LIN {X 0,Y 518.293,Z 267.839,A -85,B 0,C 180,E1 -4920.11,E2 -4920.11} C_VEL
LIN {X 0,Y 518.366,Z 255.687,A -85,B 0,C 180,E1 -4920.557,E2 -4920.557} C_VEL
LIN {X 0,Y 516.298,Z 245.529,A -85,B 0,C 180,E1 -4920.881,E2 -4920.881} C_VEL
LIN {X 0,Y 516.387,Z 241.725,A -85,B 0,C 180,E1 -4924.182,E2 -4924.182} C_VEL
LIN {X 0,Y 516.405,Z 238.771,A -85,B 0,C 180,E1 -4926.755,E2 -4926.755} C_VEL
LIN {X 0,Y 516.418,Z 234.973,A -85,B 0,C 180,E1 -4930.11,E2 -4930.11} C_VEL
LIN {X 0,Y 516.464,Z 232.179,A -85,B 0,C 180,E1 -4932.581,E2 -4932.581} C_VEL
LIN {X 0,Y 516.496,Z 228.529,A -85,B 0,C 180,E1 -4935.823,E2 -4935.823} C_VEL
LIN {X 0,Y 516.609,Z 224.947,A -85,B 0,C 180,E1 -4939.021,E2 -4939.021} C_VEL
LIN {X 0,Y 516.557,Z 224.144,A -85,B 0,C 180,E1 -4939.813,E2 -4939.813} C_VEL
LIN {X 0,Y 516.894,Z 224.101,A -85,B 0,C 180,E1 -4942.186,E2 -4942.186} C_VEL
LIN {X 0,Y 517.03,Z 224.083,A -85,B 0,C 180,E1 -4944.54,E2 -4944.54} C_VEL
LIN {X 0,Y 517.069,Z 224.078,A -85,B 0,C 180,E1 -4947.664,E2 -4947.664} C_VEL
LIN {X 0,Y 517.082,Z 224.079,A -85,B 0,C 180,E1 -4950.779,E2 -4950.779} C_VEL
LIN {X 0,Y 517.001,Z 224.089,A -85,B 0,C 180,E1 -4953.117,E2 -4953.117} C_VEL
LIN {X 0,Y 516.996,Z 224.086,A -85,B 0,C 180,E1 -4956.244,E2 -4956.244} C_VEL
LIN {X 0,Y 516.943,Z 224.094,A -85,B 0,C 180,E1 -4959.39,E2 -4959.39} C_VEL
LIN {X 0,Y 516.967,Z 224.089,A -85,B 0,C 180,E1 -4961.825,E2 -4961.825} C_VEL
LIN {X 0,Y 516.928,Z 224.097,A -85,B 0,C 180,E1 -4965.147,E2 -4965.147} C_VEL
LIN {X 0,Y 516.912,Z 224.097,A -85,B 0,C 180,E1 -4968.223,E2 -4968.223} C_VEL
LIN {X 0,Y 516.902,Z 224.1,A -85,B 0,C 180,E1 -4970.702,E2 -4970.702} C_VEL
LIN {X 0,Y 516.881,Z 224.104,A -85,B 0,C 180,E1 -4973.223,E2 -4973.223} C_VEL
LIN {X 0,Y 516.932,Z 224.095,A -85,B 0,C 180,E1 -4976.198,E2 -4976.198} C_VEL
LIN {X 0,Y 516.909,Z 224.099,A -85,B 0,C 180,E1 -4979.306,E2 -4979.306} C_VEL
LIN {X 0,Y 516.889,Z 224.101,A -85,B 0,C 180,E1 -4982.546,E2 -4982.546} C_VEL
LIN {X 0,Y 516.871,Z 224.103,A -85,B 0,C 180,E1 -4985.334,E2 -4985.334} C_VEL
LIN {X 0,Y 516.871,Z 224.103,A -85,B 0,C 180,E1 -4987.945,E2 -4987.945} C_VEL
LIN {X 0,Y 516.898,Z 224.1,A -85,B 0,C 180,E1 -4990.741,E2 -4990.741} C_VEL
LIN {X 0,Y 516.873,Z 224.103,A -85,B 0,C 180,E1 -4993.904,E2 -4993.904} C_VEL
LIN {X 0,Y 516.873,Z 224.104,A -85,B 0,C 180,E1 -4996.108,E2 -4996.108} C_VEL
LIN {X 0,Y 516.896,Z 224.101,A -85,B 0,C 180,E1 -4999.262,E2 -4999.262} C_VEL
LIN {X 0,Y 516.875,Z 224.104,A -85,B 0,C 180,E1 -5002.058,E2 -5002.058} C_VEL
LIN {X 0,Y 516.888,Z 224.101,A -85,B 0,C 180,E1 -5005.178,E2 -5005.178} C_VEL
LIN {X 0,Y 516.878,Z 224.104,A -85,B 0,C 180,E1 -5007.977,E2 -5007.977} C_VEL
LIN {X 0,Y 516.932,Z 224.095,A -85,B 0,C 180,E1 -5010.698,E2 -5010.698} C_VEL
LIN {X 0,Y 516.939,Z 224.096,A -85,B 0,C 180,E1 -5013.805,E2 -5013.805} C_VEL
LIN {X 0,Y 516.869,Z 224.102,A -85,B 0,C 180,E1 -5016.778,E2 -5016.778} C_VEL
LIN {X 0,Y 516.937,Z 224.096,A -85,B 0,C 180,E1 -5019.733,E2 -5019.733} C_VEL
LIN {X 0,Y 516.93,Z 224.095,A -85,B 0,C 180,E1 -5022.598,E2 -5022.598} C_VEL
LIN {X 0,Y 516.941,Z 224.093,A -85,B 0,C 180,E1 -5025.032,E2 -5025.032} C_VEL
LIN {X 0,Y 516.966,Z 224.092,A -85,B 0,C 180,E1 -5028.235,E2 -5028.235} C_VEL
LIN {X 0,Y 516.955,Z 224.092,A -85,B 0,C 180,E1 -5031.401,E2 -5031.401} C_VEL
LIN {X 0,Y 517.011,Z 224.086,A -85,B 0,C 180,E1 -5033.758,E2 -5033.758} C_VEL
LIN {X 0,Y 517.082,Z 224.079,A -85,B 0,C 180,E1 -5037.664,E2 -5037.664} C_VEL
LIN {X 0,Y 517.094,Z 224.074,A -85,B 0,C 180,E1 -5040.78,E2 -5040.78} C_VEL
LIN {X 0,Y 517.013,Z 224.084,A -85,B 0,C 180,E1 -5043.118,E2 -5043.118} C_VEL
LIN {X 0,Y 516.992,Z 224.087,A -85,B 0,C 180,E1 -5046.245,E2 -5046.245} C_VEL
LIN {X 0,Y 516.945,Z 224.095,A -85,B 0,C 180,E1 -5049.391,E2 -5049.391} C_VEL
LIN {X 0,Y 516.956,Z 224.094,A -85,B 0,C 180,E1 -5051.808,E2 -5051.808} C_VEL
LIN {X 0,Y 516.95,Z 224.093,A -85,B 0,C 180,E1 -5055.147,E2 -5055.147} C_VEL
LIN {X 0,Y 516.93,Z 224.094,A -85,B 0,C 180,E1 -5058.223,E2 -5058.223} C_VEL
LIN {X 0,Y 516.918,Z 224.097,A -85,B 0,C 180,E1 -5060.702,E2 -5060.702} C_VEL
LIN {X 0,Y 516.891,Z 224.1,A -85,B 0,C 180,E1 -5064.074,E2 -5064.074} C_VEL
LIN {X 0,Y 516.915,Z 224.097,A -85,B 0,C 180,E1 -5066.659,E2 -5066.659} C_VEL
LIN {X 0,Y 516.915,Z 224.098,A -85,B 0,C 180,E1 -5069.524,E2 -5069.524} C_VEL
LIN {X 0,Y 516.9,Z 224.099,A -85,B 0,C 180,E1 -5072.544,E2 -5072.544} C_VEL
LIN {X 0,Y 516.872,Z 224.103,A -85,B 0,C 180,E1 -5075.33,E2 -5075.33} C_VEL
LIN {X 0,Y 516.886,Z 224.102,A -85,B 0,C 180,E1 -5077.943,E2 -5077.943} C_VEL
LIN {X 0,Y 516.889,Z 224.102,A -85,B 0,C 180,E1 -5080.742,E2 -5080.742} C_VEL
LIN {X 0,Y 516.888,Z 224.101,A -85,B 0,C 180,E1 -5082.832,E2 -5082.832} C_VEL
LIN {X 0,Y 516.901,Z 224.098,A -85,B 0,C 180,E1 -5085.007,E2 -5085.007} C_VEL
LIN {X 0,Y 516.919,Z 224.097,A -85,B 0,C 180,E1 -5088.399,E2 -5088.399} C_VEL
LIN {X 0,Y 516.919,Z 224.183,A -85,B 0,C 180,E1 -5091.168,E2 -5091.168} C_VEL
LIN {X 0,Y 518.071,Z 230.899,A -85,B 0,C 180,E1 -5093.835,E2 -5093.835} C_VEL
LIN {X 0,Y 518.092,Z 236.578,A -85,B 0,C 180,E1 -5095.841,E2 -5095.841} C_VEL
LIN {X 0,Y 517.808,Z 245.682,A -85,B 0,C 180,E1 -5098.952,E2 -5098.952} C_VEL
LIN {X 0,Y 517.592,Z 254.692,A -85,B 0,C 180,E1 -5101.957,E2 -5101.957} C_VEL
LIN {X 0,Y 517.295,Z 264.28,A -85,B 0,C 180,E1 -5105.091,E2 -5105.091} C_VEL
LIN {X 0,Y 517.075,Z 273.548,A -85,B 0,C 180,E1 -5108.051,E2 -5108.051} C_VEL
LIN {X 0,Y 516.883,Z 282.815,A -85,B 0,C 180,E1 -5110.954,E2 -5110.954} C_VEL
LIN {X 0,Y 516.697,Z 292.082,A -85,B 0,C 180,E1 -5113.809,E2 -5113.809} C_VEL
LIN {X 0,Y 516.588,Z 299.708,A -85,B 0,C 180,E1 -5116.095,E2 -5116.095} C_VEL
LIN {X 0,Y 518.517,Z 312.169,A -85,B 0,C 180,E1 -5116.428,E2 -5116.428} C_VEL
LIN {X 0,Y 518.247,Z 324.975,A -85,B 0,C 180,E1 -5116.87,E2 -5116.87} C_VEL
LIN {X 0,Y 517.941,Z 337.168,A -85,B 0,C 180,E1 -5117.461,E2 -5117.461} C_VEL
LIN {X 0,Y 517.619,Z 349.582,A -85,B 0,C 180,E1 -5118.248,E2 -5118.248} C_VEL
LIN {X 0,Y 517.326,Z 360.466,A -85,B 0,C 180,E1 -5119.135,E2 -5119.135} C_VEL
LIN {X 0,Y 517.045,Z 369.331,A -85,B 0,C 180,E1 -5120.02,E2 -5120.02} C_VEL
LIN {X 0,Y 516.813,Z 378.958,A -85,B 0,C 180,E1 -5121.2,E2 -5121.2} C_VEL
LIN {X 0,Y 516.565,Z 386.619,A -85,B 0,C 180,E1 -5122.377,E2 -5122.377} C_VEL
LIN {X 0,Y 516.428,Z 393.678,A -85,B 0,C 180,E1 -5123.749,E2 -5123.749} C_VEL
LIN {X 0,Y 516.314,Z 398.371,A -85,B 0,C 180,E1 -5124.924,E2 -5124.924} C_VEL
LIN {X 0,Y 516.355,Z 401.957,A -85,B 0,C 180,E1 -5126.097,E2 -5126.097} C_VEL
LIN {X 0,Y 516.283,Z 403.807,A -85,B 0,C 180,E1 -5126.878,E2 -5126.878} C_VEL
LIN {X 0,Y 516.262,Z 405.196,A -85,B 0,C 180,E1 -5127.659,E2 -5127.659} C_VEL
LIN {X 0,Y 516.16,Z 406.785,A -85,B 0,C 180,E1 -5129.219,E2 -5129.219} C_VEL
LIN {X 0,Y 516.154,Z 407,A -85,B 0,C 180,E1 -5130,E2 -5130} C_VEL
LIN {X 0,Y 516.192,Z 406.186,A -85,B 0,C 180,E1 -5131.56,E2 -5131.56} C_VEL
LIN {X 0,Y 516.262,Z 405.199,A -85,B 0,C 180,E1 -5132.34,E2 -5132.34} C_VEL
LIN {X 0,Y 516.283,Z 403.811,A -85,B 0,C 180,E1 -5133.121,E2 -5133.121} C_VEL
LIN {X 0,Y 516.344,Z 400.897,A -85,B 0,C 180,E1 -5134.293,E2 -5134.293} C_VEL
LIN {X 0,Y 516.406,Z 396.95,A -85,B 0,C 180,E1 -5135.466,E2 -5135.466} C_VEL
LIN {X 0,Y 516.487,Z 391.037,A -85,B 0,C 180,E1 -5136.807,E2 -5136.807} C_VEL
LIN {X 0,Y 516.642,Z 384.24,A -85,B 0,C 180,E1 -5138.015,E2 -5138.015} C_VEL
LIN {X 0,Y 516.868,Z 375.995,A -85,B 0,C 180,E1 -5139.193,E2 -5139.193} C_VEL
LIN {X 0,Y 517.079,Z 367.544,A -85,B 0,C 180,E1 -5140.177,E2 -5140.177} C_VEL
LIN {X 0,Y 517.455,Z 357.102,A -85,B 0,C 180,E1 -5141.159,E2 -5141.159} C_VEL
LIN {X 0,Y 517.7,Z 345.79,A -85,B 0,C 180,E1 -5142.015,E2 -5142.015} C_VEL
LIN {X 0,Y 518,Z 335.417,A -85,B 0,C 180,E1 -5142.637,E2 -5142.637} C_VEL
LIN {X 0,Y 518.28,Z 323.777,A -85,B 0,C 180,E1 -5143.178,E2 -5143.178} C_VEL
LIN {X 0,Y 518.371,Z 310.365,A -85,B 0,C 180,E1 -5143.625,E2 -5143.625} C_VEL
LIN {X 0,Y 516.57,Z 299.532,A -85,B 0,C 180,E1 -5143.924,E2 -5143.924} C_VEL
LIN {X 0,Y 516.712,Z 290.761,A -85,B 0,C 180,E1 -5146.596,E2 -5146.596} C_VEL
LIN {X 0,Y 516.906,Z 281.494,A -85,B 0,C 180,E1 -5149.457,E2 -5149.457} C_VEL
LIN {X 0,Y 517.099,Z 271.966,A -85,B 0,C 180,E1 -5152.45,E2 -5152.45} C_VEL
LIN {X 0,Y 517.322,Z 262.959,A -85,B 0,C 180,E1 -5155.336,E2 -5155.336} C_VEL
LIN {X 0,Y 517.601,Z 253.641,A -85,B 0,C 180,E1 -5158.374,E2 -5158.374} C_VEL
LIN {X 0,Y 517.835,Z 244.076,A -85,B 0,C 180,E1 -5161.547,E2 -5161.547} C_VEL
LIN {X 0,Y 518.14,Z 234.767,A -85,B 0,C 180,E1 -5164.727,E2 -5164.727} C_VEL
LIN {X 0,Y 518.063,Z 230.835,A -85,B 0,C 180,E1 -5166.165,E2 -5166.165} C_VEL
LIN {X 0,Y 516.897,Z 224.101,A -85,B 0,C 180,E1 -5168.892,E2 -5168.892} C_VEL
LIN {X 0,Y 516.913,Z 224.1,A -85,B 0,C 180,E1 -5171.774,E2 -5171.774} C_VEL
LIN {X 0,Y 516.924,Z 224.097,A -85,B 0,C 180,E1 -5175.009,E2 -5175.009} C_VEL
LIN {X 0,Y 516.924,Z 224.097,A -85,B 0,C 180,E1 -5178.397,E2 -5178.397} C_VEL
LIN {X 0,Y 516.887,Z 224.102,A -85,B 0,C 180,E1 -5181.284,E2 -5181.284} C_VEL
LIN {X 0,Y 516.871,Z 224.104,A -85,B 0,C 180,E1 -5184.219,E2 -5184.219} C_VEL
LIN {X 0,Y 516.894,Z 224.102,A -85,B 0,C 180,E1 -5187.052,E2 -5187.052} C_VEL
LIN {X 0,Y 516.892,Z 224.101,A -85,B 0,C 180,E1 -5189.795,E2 -5189.795} C_VEL
LIN {X 0,Y 516.93,Z 224.096,A -85,B 0,C 180,E1 -5192.466,E2 -5192.466} C_VEL
LIN {X 0,Y 516.912,Z 224.098,A -85,B 0,C 180,E1 -5195.071,E2 -5195.071} C_VEL
LIN {X 0,Y 516.886,Z 224.103,A -85,B 0,C 180,E1 -5198.461,E2 -5198.461} C_VEL
LIN {X 0,Y 516.903,Z 224.099,A -85,B 0,C 180,E1 -5200.954,E2 -5200.954} C_VEL
LIN {X 0,Y 516.914,Z 224.098,A -85,B 0,C 180,E1 -5203.409,E2 -5203.409} C_VEL
LIN {X 0,Y 516.894,Z 224.102,A -85,B 0,C 180,E1 -5205.832,E2 -5205.832} C_VEL
LIN {X 0,Y 516.963,Z 224.092,A -85,B 0,C 180,E1 -5208.232,E2 -5208.232} C_VEL
LIN {X 0,Y 516.967,Z 224.09,A -85,B 0,C 180,E1 -5211.398,E2 -5211.398} C_VEL
LIN {X 0,Y 517.009,Z 224.085,A -85,B 0,C 180,E1 -5213.756,E2 -5213.756} C_VEL
LIN {X 0,Y 517.081,Z 224.076,A -85,B 0,C 180,E1 -5217.662,E2 -5217.662} C_VEL
LIN {X 0,Y 517.092,Z 224.076,A -85,B 0,C 180,E1 -5220.777,E2 -5220.777} C_VEL
LIN {X 0,Y 517.01,Z 224.086,A -85,B 0,C 180,E1 -5223.116,E2 -5223.116} C_VEL
LIN {X 0,Y 517.005,Z 224.087,A -85,B 0,C 180,E1 -5226.242,E2 -5226.242} C_VEL
LIN {X 0,Y 516.951,Z 224.094,A -85,B 0,C 180,E1 -5229.388,E2 -5229.388} C_VEL
LIN {X 0,Y 516.871,Z 224.108,A -85,B 0,C 180,E1 -5231.767,E2 -5231.767} C_VEL
LIN {X 0,Y 516.656,Z 224.134,A -85,B 0,C 180,E1 -5233.369,E2 -5233.369} C_VEL
LIN {X 0,Y 516.611,Z 226.687,A -85,B 0,C 180,E1 -5235.787,E2 -5235.787} C_VEL
LIN {X 0,Y 516.586,Z 229.392,A -85,B 0,C 180,E1 -5238.233,E2 -5238.233} C_VEL
LIN {X 0,Y 516.503,Z 232.073,A -85,B 0,C 180,E1 -5240.717,E2 -5240.717} C_VEL
LIN {X 0,Y 516.477,Z 234.853,A -85,B 0,C 180,E1 -5243.24,E2 -5243.24} C_VEL
LIN {X 0,Y 516.443,Z 237.987,A -85,B 0,C 180,E1 -5246.084,E2 -5246.084} C_VEL
LIN {X 0,Y 516.356,Z 240.593,A -85,B 0,C 180,E1 -5248.447,E2 -5248.447} C_VEL
LIN {X 0,Y 516.337,Z 243.593,A -85,B 0,C 180,E1 -5251.144,E2 -5251.144} C_VEL
LIN {X 0,Y 516.326,Z 245.939,A -85,B 0,C 180,E1 -5253.219,E2 -5253.219} C_VEL
LIN {X 0,Y 518.499,Z 256.466,A -85,B 0,C 180,E1 -5253.555,E2 -5253.555} C_VEL
LIN {X 0,Y 518.309,Z 269.575,A -85,B 0,C 180,E1 -5254.049,E2 -5254.049} C_VEL
LIN {X 0,Y 517.979,Z 281.539,A -85,B 0,C 180,E1 -5254.661,E2 -5254.661} C_VEL
LIN {X 0,Y 517.683,Z 292.312,A -85,B 0,C 180,E1 -5255.375,E2 -5255.375} C_VEL
LIN {X 0,Y 517.421,Z 302.46,A -85,B 0,C 180,E1 -5256.215,E2 -5256.215} C_VEL
LIN {X 0,Y 517.109,Z 312.236,A -85,B 0,C 180,E1 -5257.211,E2 -5257.211} C_VEL
LIN {X 0,Y 516.846,Z 320.928,A -85,B 0,C 180,E1 -5258.304,E2 -5258.304} C_VEL
LIN {X 0,Y 516.673,Z 328.117,A -85,B 0,C 180,E1 -5259.424,E2 -5259.424} C_VEL
LIN {X 0,Y 516.46,Z 335.038,A -85,B 0,C 180,E1 -5260.78,E2 -5260.78} C_VEL
LIN {X 0,Y 516.409,Z 339.222,A -85,B 0,C 180,E1 -5261.823,E2 -5261.823} C_VEL
LIN {X 0,Y 516.376,Z 342.593,A -85,B 0,C 180,E1 -5262.881,E2 -5262.881} C_VEL
LIN {X 0,Y 516.299,Z 345.203,A -85,B 0,C 180,E1 -5263.963,E2 -5263.963} C_VEL
LIN {X 0,Y 516.245,Z 346.43,A -85,B 0,C 180,E1 -5264.701,E2 -5264.701} C_VEL
LIN {X 0,Y 515.559,Z 347.393,A -85,B 0,C 180,E1 -5265.343,E2 -5265.343} C_VEL
LIN {X 0,Y 512.637,Z 348.352,A -85,B 0,C 180,E1 -5266.394,E2 -5266.394} C_VEL
LIN {X 0,Y 510.196,Z 348.597,A -85,B 0,C 180,E1 -5267.245,E2 -5267.245} C_VEL
LIN {X 0,Y 509.183,Z 348.434,A -85,B 0,C 180,E1 -5267.903,E2 -5267.903} C_VEL
LIN {X 0,Y 509.12,Z 348.292,A -85,B 0,C 180,E1 -5268.125,E2 -5268.125} C_VEL
LIN {X 0,Y 509.192,Z 346.685,A -85,B 0,C 180,E1 -5269.557,E2 -5269.557} C_VEL
LIN {X 0,Y 509.266,Z 343.364,A -85,B 0,C 180,E1 -5271.114,E2 -5271.114} C_VEL
LIN {X 0,Y 509.355,Z 338.563,A -85,B 0,C 180,E1 -5272.62,E2 -5272.62} C_VEL
LIN {X 0,Y 509.507,Z 333.29,A -85,B 0,C 180,E1 -5273.847,E2 -5273.847} C_VEL
LIN {X 0,Y 509.684,Z 326.491,A -85,B 0,C 180,E1 -5275.094,E2 -5275.094} C_VEL
LIN {X 0,Y 509.95,Z 318.211,A -85,B 0,C 180,E1 -5276.31,E2 -5276.31} C_VEL
LIN {X 0,Y 510.231,Z 309.563,A -85,B 0,C 180,E1 -5277.339,E2 -5277.339} C_VEL
LIN {X 0,Y 510.538,Z 299.077,A -85,B 0,C 180,E1 -5278.344,E2 -5278.344} C_VEL
LIN {X 0,Y 510.883,Z 288.287,A -85,B 0,C 180,E1 -5279.175,E2 -5279.175} C_VEL
LIN {X 0,Y 511.163,Z 277.602,A -85,B 0,C 180,E1 -5279.831,E2 -5279.831} C_VEL
LIN {X 0,Y 511.471,Z 265.262,A -85,B 0,C 180,E1 -5280.409,E2 -5280.409} C_VEL
LIN {X 0,Y 511.37,Z 256.106,A -85,B 0,C 180,E1 -5280.742,E2 -5280.742} C_VEL
LIN {X 0,Y 509.241,Z 245.892,A -85,B 0,C 180,E1 -5281.089,E2 -5281.089} C_VEL
LIN {X 0,Y 509.301,Z 242.78,A -85,B 0,C 180,E1 -5283.796,E2 -5283.796} C_VEL
LIN {X 0,Y 509.3,Z 239.785,A -85,B 0,C 180,E1 -5286.411,E2 -5286.411} C_VEL
LIN {X 0,Y 509.336,Z 236.004,A -85,B 0,C 180,E1 -5289.76,E2 -5289.76} C_VEL
LIN {X 0,Y 509.407,Z 233.109,A -85,B 0,C 180,E1 -5292.331,E2 -5292.331} C_VEL
LIN {X 0,Y 509.438,Z 229.427,A -85,B 0,C 180,E1 -5295.622,E2 -5295.622} C_VEL
LIN {X 0,Y 509.541,Z 225.808,A -85,B 0,C 180,E1 -5298.867,E2 -5298.867} C_VEL
LIN {X 0,Y 509.512,Z 225.022,A -85,B 0,C 180,E1 -5299.671,E2 -5299.671} C_VEL
LIN {X 0,Y 509.837,Z 224.98,A -85,B 0,C 180,E1 -5302.077,E2 -5302.077} C_VEL
LIN {X 0,Y 509.979,Z 224.961,A -85,B 0,C 180,E1 -5304.465,E2 -5304.465} C_VEL
LIN {X 0,Y 510.04,Z 224.954,A -85,B 0,C 180,E1 -5307.631,E2 -5307.631} C_VEL
LIN {X 0,Y 510.038,Z 224.953,A -85,B 0,C 180,E1 -5310,E2 -5310} C_VEL
LIN {X 0,Y 510.041,Z 224.952,A -85,B 0,C 180,E1 -5312.37,E2 -5312.37} C_VEL
LIN {X 0,Y 509.964,Z 224.963,A -85,B 0,C 180,E1 -5316.33,E2 -5316.33} C_VEL
LIN {X 0,Y 509.904,Z 224.971,A -85,B 0,C 180,E1 -5318.721,E2 -5318.721} C_VEL
LIN {X 0,Y 509.935,Z 224.965,A -85,B 0,C 180,E1 -5321.931,E2 -5321.931} C_VEL
LIN {X 0,Y 509.878,Z 224.974,A -85,B 0,C 180,E1 -5325.243,E2 -5325.243} C_VEL
LIN {X 0,Y 509.874,Z 224.973,A -85,B 0,C 180,E1 -5328.002,E2 -5328.002} C_VEL
LIN {X 0,Y 509.846,Z 224.98,A -85,B 0,C 180,E1 -5331.002,E2 -5331.002} C_VEL
LIN {X 0,Y 509.839,Z 224.978,A -85,B 0,C 180,E1 -5333.563,E2 -5333.563} C_VEL
LIN {X 0,Y 509.9,Z 224.971,A -85,B 0,C 180,E1 -5336.38,E2 -5336.38} C_VEL
LIN {X 0,Y 509.864,Z 224.976,A -85,B 0,C 180,E1 -5338.845,E2 -5338.845} C_VEL
LIN {X 0,Y 509.813,Z 224.983,A -85,B 0,C 180,E1 -5341.591,E2 -5341.591} C_VEL
LIN {X 0,Y 509.842,Z 224.979,A -85,B 0,C 180,E1 -5344.414,E2 -5344.414} C_VEL
LIN {X 0,Y 509.808,Z 224.984,A -85,B 0,C 180,E1 -5347.342,E2 -5347.342} C_VEL
LIN {X 0,Y 509.853,Z 224.977,A -85,B 0,C 180,E1 -5350.381,E2 -5350.381} C_VEL
LIN {X 0,Y 509.831,Z 224.98,A -85,B 0,C 180,E1 -5353.066,E2 -5353.066} C_VEL
LIN {X 0,Y 509.821,Z 224.981,A -85,B 0,C 180,E1 -5355.794,E2 -5355.794} C_VEL
LIN {X 0,Y 509.857,Z 224.977,A -85,B 0,C 180,E1 -5358.577,E2 -5358.577} C_VEL
LIN {X 0,Y 509.851,Z 224.977,A -85,B 0,C 180,E1 -5361.664,E2 -5361.664} C_VEL
LIN {X 0,Y 509.838,Z 224.979,A -85,B 0,C 180,E1 -5364.625,E2 -5364.625} C_VEL
LIN {X 0,Y 509.861,Z 224.975,A -85,B 0,C 180,E1 -5367.483,E2 -5367.483} C_VEL
LIN {X 0,Y 509.877,Z 224.976,A -85,B 0,C 180,E1 -5370.271,E2 -5370.271} C_VEL
LIN {X 0,Y 509.881,Z 224.972,A -85,B 0,C 180,E1 -5372.946,E2 -5372.946} C_VEL
LIN {X 0,Y 509.866,Z 224.975,A -85,B 0,C 180,E1 -5375.576,E2 -5375.576} C_VEL
LIN {X 0,Y 509.82,Z 224.981,A -85,B 0,C 180,E1 -5378.15,E2 -5378.15} C_VEL
LIN {X 0,Y 509.863,Z 224.977,A -85,B 0,C 180,E1 -5380.683,E2 -5380.683} C_VEL
LIN {X 0,Y 509.886,Z 224.973,A -85,B 0,C 180,E1 -5383.176,E2 -5383.176} C_VEL
LIN {X 0,Y 509.863,Z 224.977,A -85,B 0,C 180,E1 -5385.636,E2 -5385.636} C_VEL
LIN {X 0,Y 509.913,Z 224.969,A -85,B 0,C 180,E1 -5388.876,E2 -5388.876} C_VEL
LIN {X 0,Y 509.921,Z 224.969,A -85,B 0,C 180,E1 -5392.079,E2 -5392.079} C_VEL
LIN {X 0,Y 509.983,Z 224.96,A -85,B 0,C 180,E1 -5394.466,E2 -5394.466} C_VEL
LIN {X 0,Y 510.054,Z 224.954,A -85,B 0,C 180,E1 -5397.632,E2 -5397.632} C_VEL
LIN {X 0,Y 510.059,Z 224.953,A -85,B 0,C 180,E1 -5400.001,E2 -5400.001} C_VEL
LIN {X 0,Y 510.055,Z 224.953,A -85,B 0,C 180,E1 -5402.37,E2 -5402.37} C_VEL
LIN {X 0,Y 509.978,Z 224.962,A -85,B 0,C 180,E1 -5405.537,E2 -5405.537} C_VEL
LIN {X 0,Y 509.908,Z 224.97,A -85,B 0,C 180,E1 -5408.722,E2 -5408.722} C_VEL
LIN {X 0,Y 509.909,Z 224.971,A -85,B 0,C 180,E1 -5411.933,E2 -5411.933} C_VEL
LIN {X 0,Y 509.899,Z 224.972,A -85,B 0,C 180,E1 -5415.243,E2 -5415.243} C_VEL
LIN {X 0,Y 509.894,Z 224.972,A -85,B 0,C 180,E1 -5418.002,E2 -5418.002} C_VEL
LIN {X 0,Y 509.856,Z 224.976,A -85,B 0,C 180,E1 -5421.003,E2 -5421.003} C_VEL
LIN {X 0,Y 509.825,Z 224.981,A -85,B 0,C 180,E1 -5423.565,E2 -5423.565} C_VEL
LIN {X 0,Y 509.892,Z 224.973,A -85,B 0,C 180,E1 -5426.373,E2 -5426.373} C_VEL
LIN {X 0,Y 509.881,Z 224.975,A -85,B 0,C 180,E1 -5428.845,E2 -5428.845} C_VEL
LIN {X 0,Y 509.824,Z 224.98,A -85,B 0,C 180,E1 -5431.591,E2 -5431.591} C_VEL
LIN {X 0,Y 509.844,Z 224.978,A -85,B 0,C 180,E1 -5434.415,E2 -5434.415} C_VEL
LIN {X 0,Y 509.823,Z 224.981,A -85,B 0,C 180,E1 -5437.341,E2 -5437.341} C_VEL
LIN {X 0,Y 509.844,Z 224.979,A -85,B 0,C 180,E1 -5440.383,E2 -5440.383} C_VEL
LIN {X 0,Y 509.829,Z 224.98,A -85,B 0,C 180,E1 -5443.062,E2 -5443.062} C_VEL
LIN {X 0,Y 509.828,Z 224.979,A -85,B 0,C 180,E1 -5445.794,E2 -5445.794} C_VEL
LIN {X 0,Y 509.861,Z 224.977,A -85,B 0,C 180,E1 -5448.575,E2 -5448.575} C_VEL
LIN {X 0,Y 509.879,Z 225.132,A -85,B 0,C 180,E1 -5450.905,E2 -5450.905} C_VEL
LIN {X 0,Y 511.088,Z 232.132,A -85,B 0,C 180,E1 -5453.751,E2 -5453.751} C_VEL
LIN {X 0,Y 511.122,Z 237.489,A -85,B 0,C 180,E1 -5455.684,E2 -5455.684} C_VEL
LIN {X 0,Y 510.854,Z 245.703,A -85,B 0,C 180,E1 -5458.536,E2 -5458.536} C_VEL
LIN {X 0,Y 510.591,Z 255.23,A -85,B 0,C 180,E1 -5461.755,E2 -5461.755} C_VEL
LIN {X 0,Y 510.303,Z 264.28,A -85,B 0,C 180,E1 -5464.726,E2 -5464.726} C_VEL
LIN {X 0,Y 510.084,Z 273.672,A -85,B 0,C 180,E1 -5467.774,E2 -5467.774} C_VEL
LIN {X 0,Y 509.861,Z 282.815,A -85,B 0,C 180,E1 -5470.681,E2 -5470.681} C_VEL
LIN {X 0,Y 509.649,Z 293.406,A -85,B 0,C 180,E1 -5473.99,E2 -5473.99} C_VEL
LIN {X 0,Y 509.541,Z 299.708,A -85,B 0,C 180,E1 -5475.898,E2 -5475.898} C_VEL
LIN {X 0,Y 511.548,Z 312.169,A -85,B 0,C 180,E1 -5476.24,E2 -5476.24} C_VEL
LIN {X 0,Y 511.335,Z 324.975,A -85,B 0,C 180,E1 -5476.69,E2 -5476.69} C_VEL
LIN {X 0,Y 511.014,Z 337.167,A -85,B 0,C 180,E1 -5477.288,E2 -5477.288} C_VEL
LIN {X 0,Y 510.744,Z 347.843,A -85,B 0,C 180,E1 -5477.964,E2 -5477.964} C_VEL
LIN {X 0,Y 510.45,Z 358.258,A -85,B 0,C 180,E1 -5478.785,E2 -5478.785} C_VEL
LIN {X 0,Y 510.072,Z 367.535,A -85,B 0,C 180,E1 -5479.681,E2 -5479.681} C_VEL
LIN {X 0,Y 509.847,Z 375.988,A -85,B 0,C 180,E1 -5480.678,E2 -5480.678} C_VEL
LIN {X 0,Y 509.586,Z 384.234,A -85,B 0,C 180,E1 -5481.873,E2 -5481.873} C_VEL
LIN {X 0,Y 509.421,Z 390.875,A -85,B 0,C 180,E1 -5483.066,E2 -5483.066} C_VEL
LIN {X 0,Y 509.345,Z 396.948,A -85,B 0,C 180,E1 -5484.457,E2 -5484.457} C_VEL
LIN {X 0,Y 509.234,Z 400.894,A -85,B 0,C 180,E1 -5485.646,E2 -5485.646} C_VEL
LIN {X 0,Y 509.201,Z 403.807,A -85,B 0,C 180,E1 -5486.835,E2 -5486.835} C_VEL
LIN {X 0,Y 509.162,Z 405.195,A -85,B 0,C 180,E1 -5487.626,E2 -5487.626} C_VEL
LIN {X 0,Y 509.074,Z 406.785,A -85,B 0,C 180,E1 -5489.209,E2 -5489.209} C_VEL
LIN {X 0,Y 509.066,Z 407,A -85,B 0,C 180,E1 -5490,E2 -5490} C_VEL
LIN {X 0,Y 509.113,Z 406.186,A -85,B 0,C 180,E1 -5491.582,E2 -5491.582} C_VEL
LIN {X 0,Y 509.162,Z 405.198,A -85,B 0,C 180,E1 -5492.373,E2 -5492.373} C_VEL
LIN {X 0,Y 509.201,Z 403.811,A -85,B 0,C 180,E1 -5493.164,E2 -5493.164} C_VEL
LIN {X 0,Y 509.234,Z 400.897,A -85,B 0,C 180,E1 -5494.353,E2 -5494.353} C_VEL
LIN {X 0,Y 509.345,Z 396.95,A -85,B 0,C 180,E1 -5495.542,E2 -5495.542} C_VEL
LIN {X 0,Y 509.411,Z 391.284,A -85,B 0,C 180,E1 -5496.853,E2 -5496.853} C_VEL
LIN {X 0,Y 509.586,Z 384.239,A -85,B 0,C 180,E1 -5498.126,E2 -5498.126} C_VEL
LIN {X 0,Y 509.847,Z 375.995,A -85,B 0,C 180,E1 -5499.321,E2 -5499.321} C_VEL
LIN {X 0,Y 510.071,Z 367.544,A -85,B 0,C 180,E1 -5500.318,E2 -5500.318} C_VEL
LIN {X 0,Y 510.478,Z 357.101,A -85,B 0,C 180,E1 -5501.314,E2 -5501.314} C_VEL
LIN {X 0,Y 510.733,Z 346.524,A -85,B 0,C 180,E1 -5502.13,E2 -5502.13} C_VEL
LIN {X 0,Y 511.06,Z 335.416,A -85,B 0,C 180,E1 -5502.811,E2 -5502.811} C_VEL
LIN {X 0,Y 511.376,Z 323.777,A -85,B 0,C 180,E1 -5503.359,E2 -5503.359} C_VEL
LIN {X 0,Y 511.458,Z 311.279,A -85,B 0,C 180,E1 -5503.787,E2 -5503.787} C_VEL
LIN {X 0,Y 509.529,Z 299.532,A -85,B 0,C 180,E1 -5504.12,E2 -5504.12} C_VEL
LIN {X 0,Y 509.718,Z 289.437,A -85,B 0,C 180,E1 -5507.243,E2 -5507.243} C_VEL
LIN {X 0,Y 509.924,Z 280.17,A -85,B 0,C 180,E1 -5510.154,E2 -5510.154} C_VEL
LIN {X 0,Y 510.121,Z 270.903,A -85,B 0,C 180,E1 -5513.119,E2 -5513.119} C_VEL
LIN {X 0,Y 510.37,Z 261.574,A -85,B 0,C 180,E1 -5516.145,E2 -5516.145} C_VEL
LIN {X 0,Y 510.605,Z 253.504,A -85,B 0,C 180,E1 -5518.799,E2 -5518.799} C_VEL
LIN {X 0,Y 510.851,Z 245.422,A -85,B 0,C 180,E1 -5521.518,E2 -5521.518} C_VEL
LIN {X 0,Y 511.179,Z 235.939,A -85,B 0,C 180,E1 -5524.794,E2 -5524.794} C_VEL
LIN {X 0,Y 511.09,Z 232.052,A -85,B 0,C 180,E1 -5526.248,E2 -5526.248} C_VEL
LIN {X 0,Y 509.861,Z 224.978,A -85,B 0,C 180,E1 -5529.159,E2 -5529.159} C_VEL
LIN {X 0,Y 509.857,Z 224.979,A -85,B 0,C 180,E1 -5531.896,E2 -5531.896} C_VEL
LIN {X 0,Y 509.858,Z 224.978,A -85,B 0,C 180,E1 -5535.331,E2 -5535.331} C_VEL
LIN {X 0,Y 509.867,Z 224.977,A -85,B 0,C 180,E1 -5538.575,E2 -5538.575} C_VEL
LIN {X 0,Y 509.853,Z 224.979,A -85,B 0,C 180,E1 -5541.661,E2 -5541.661} C_VEL
LIN {X 0,Y 509.83,Z 224.982,A -85,B 0,C 180,E1 -5544.621,E2 -5544.621} C_VEL
LIN {X 0,Y 509.861,Z 224.977,A -85,B 0,C 180,E1 -5547.48,E2 -5547.48} C_VEL
LIN {X 0,Y 509.858,Z 224.977,A -85,B 0,C 180,E1 -5550.273,E2 -5550.273} C_VEL
LIN {X 0,Y 509.887,Z 224.973,A -85,B 0,C 180,E1 -5552.943,E2 -5552.943} C_VEL
LIN {X 0,Y 509.87,Z 224.975,A -85,B 0,C 180,E1 -5555.573,E2 -5555.573} C_VEL
LIN {X 0,Y 509.822,Z 224.98,A -85,B 0,C 180,E1 -5558.148,E2 -5558.148} C_VEL
LIN {X 0,Y 509.863,Z 224.977,A -85,B 0,C 180,E1 -5560.68,E2 -5560.68} C_VEL
LIN {X 0,Y 509.884,Z 224.973,A -85,B 0,C 180,E1 -5563.174,E2 -5563.174} C_VEL
LIN {X 0,Y 509.862,Z 224.978,A -85,B 0,C 180,E1 -5565.633,E2 -5565.633} C_VEL
LIN {X 0,Y 509.911,Z 224.971,A -85,B 0,C 180,E1 -5568.873,E2 -5568.873} C_VEL
LIN {X 0,Y 509.949,Z 224.967,A -85,B 0,C 180,E1 -5572.077,E2 -5572.077} C_VEL
LIN {X 0,Y 509.981,Z 224.962,A -85,B 0,C 180,E1 -5574.463,E2 -5574.463} C_VEL
LIN {X 0,Y 510.052,Z 224.951,A -85,B 0,C 180,E1 -5577.63,E2 -5577.63} C_VEL
LIN {X 0,Y 510.062,Z 224.951,A -85,B 0,C 180,E1 -5580.788,E2 -5580.788} C_VEL
LIN {X 0,Y 509.952,Z 224.965,A -85,B 0,C 180,E1 -5583.159,E2 -5583.159} C_VEL
LIN {X 0,Y 509.973,Z 224.964,A -85,B 0,C 180,E1 -5586.328,E2 -5586.328} C_VEL
LIN {X 0,Y 509.913,Z 224.972,A -85,B 0,C 180,E1 -5588.719,E2 -5588.719} C_VEL
LIN {X 0,Y 509.812,Z 224.988,A -85,B 0,C 180,E1 -5591.932,E2 -5591.932} C_VEL
LIN {X 0,Y 509.604,Z 225.018,A -85,B 0,C 180,E1 -5593.558,E2 -5593.558} C_VEL
LIN {X 0,Y 509.552,Z 227.696,A -85,B 0,C 180,E1 -5596.011,E2 -5596.011} C_VEL
LIN {X 0,Y 509.536,Z 230.422,A -85,B 0,C 180,E1 -5598.494,E2 -5598.494} C_VEL
LIN {X 0,Y 509.423,Z 233.191,A -85,B 0,C 180,E1 -5601.018,E2 -5601.018} C_VEL
LIN {X 0,Y 509.396,Z 235.921,A -85,B 0,C 180,E1 -5603.583,E2 -5603.583} C_VEL
LIN {X 0,Y 509.376,Z 238.895,A -85,B 0,C 180,E1 -5606.258,E2 -5606.258} C_VEL
LIN {X 0,Y 509.288,Z 241.774,A -85,B 0,C 180,E1 -5608.879,E2 -5608.879} C_VEL
LIN {X 0,Y 509.238,Z 244.828,A -85,B 0,C 180,E1 -5611.628,E2 -5611.628} C_VEL
LIN {X 0,Y 509.256,Z 246.375,A -85,B 0,C 180,E1 -5613.023,E2 -5613.023} C_VEL
LIN {X 0,Y 511.598,Z 257.395,A -85,B 0,C 180,E1 -5613.389,E2 -5613.389} C_VEL
LIN {X 0,Y 511.401,Z 270.077,A -85,B 0,C 180,E1 -5613.876,E2 -5613.876} C_VEL
LIN {X 0,Y 511.077,Z 281.752,A -85,B 0,C 180,E1 -5614.481,E2 -5614.481} C_VEL
LIN {X 0,Y 510.755,Z 292.327,A -85,B 0,C 180,E1 -5615.184,E2 -5615.184} C_VEL
LIN {X 0,Y 510.451,Z 303.39,A -85,B 0,C 180,E1 -5616.115,E2 -5616.115} C_VEL
LIN {X 0,Y 510.13,Z 312.939,A -85,B 0,C 180,E1 -5617.108,E2 -5617.108} C_VEL
LIN {X 0,Y 509.845,Z 321.561,A -85,B 0,C 180,E1 -5618.214,E2 -5618.214} C_VEL
LIN {X 0,Y 509.606,Z 329.225,A -85,B 0,C 180,E1 -5619.44,E2 -5619.44} C_VEL
LIN {X 0,Y 509.409,Z 335.244,A -85,B 0,C 180,E1 -5620.642,E2 -5620.642} C_VEL
LIN {X 0,Y 509.358,Z 339.955,A -85,B 0,C 180,E1 -5621.835,E2 -5621.835} C_VEL
LIN {X 0,Y 509.285,Z 343.493,A -85,B 0,C 180,E1 -5622.998,E2 -5622.998} C_VEL
LIN {X 0,Y 509.198,Z 346.029,A -85,B 0,C 180,E1 -5624.135,E2 -5624.135} C_VEL
LIN {X 0,Y 509.147,Z 347.693,A -85,B 0,C 180,E1 -5625.254,E2 -5625.254} C_VEL
LIN {X 0,Y 509.131,Z 348.549,A -85,B 0,C 180,E1 -5626.355,E2 -5626.355} C_VEL
LIN {X 0,Y 509.088,Z 348.624,A -85,B 0,C 180,E1 -5627.434,E2 -5627.434} C_VEL
LIN {X 0,Y 509.12,Z 348.292,A -85,B 0,C 180,E1 -5628.125,E2 -5628.125} C_VEL
LIN {X 0,Y 508.504,Z 347.825,A -85,B 0,C 180,E1 -5628.784,E2 -5628.784} C_VEL
LIN {X 0,Y 505.675,Z 346.46,A -85,B 0,C 180,E1 -5629.846,E2 -5629.846} C_VEL
LIN {X 0,Y 503.279,Z 344.879,A -85,B 0,C 180,E1 -5630.692,E2 -5630.692} C_VEL
LIN {X 0,Y 502.281,Z 343.339,A -85,B 0,C 180,E1 -5631.337,E2 -5631.337} C_VEL
LIN {X 0,Y 502.219,Z 342.739,A -85,B 0,C 180,E1 -5631.553,E2 -5631.553} C_VEL
LIN {X 0,Y 502.326,Z 337.726,A -85,B 0,C 180,E1 -5633.016,E2 -5633.016} C_VEL
LIN {X 0,Y 502.524,Z 331.369,A -85,B 0,C 180,E1 -5634.41,E2 -5634.41} C_VEL
LIN {X 0,Y 502.729,Z 324.692,A -85,B 0,C 180,E1 -5635.565,E2 -5635.565} C_VEL
LIN {X 0,Y 503.041,Z 316.207,A -85,B 0,C 180,E1 -5636.746,E2 -5636.746} C_VEL
LIN {X 0,Y 503.397,Z 306.491,A -85,B 0,C 180,E1 -5637.842,E2 -5637.842} C_VEL
LIN {X 0,Y 503.7,Z 296.746,A -85,B 0,C 180,E1 -5638.733,E2 -5638.733} C_VEL
LIN {X 0,Y 504.043,Z 285.952,A -85,B 0,C 180,E1 -5639.525,E2 -5639.525} C_VEL
LIN {X 0,Y 504.325,Z 274.72,A -85,B 0,C 180,E1 -5640.178,E2 -5640.178} C_VEL
LIN {X 0,Y 504.655,Z 262.511,A -85,B 0,C 180,E1 -5640.715,E2 -5640.715} C_VEL
LIN {X 0,Y 504.426,Z 256.567,A -85,B 0,C 180,E1 -5640.929,E2 -5640.929} C_VEL
LIN {X 0,Y 502.184,Z 246.288,A -85,B 0,C 180,E1 -5641.274,E2 -5641.274} C_VEL
LIN {X 0,Y 502.215,Z 242.824,A -85,B 0,C 180,E1 -5644.291,E2 -5644.291} C_VEL
LIN {X 0,Y 502.233,Z 239.24,A -85,B 0,C 180,E1 -5647.448,E2 -5647.448} C_VEL
LIN {X 0,Y 502.259,Z 235.954,A -85,B 0,C 180,E1 -5650.378,E2 -5650.378} C_VEL
LIN {X 0,Y 502.316,Z 233.112,A -85,B 0,C 180,E1 -5652.914,E2 -5652.914} C_VEL
LIN {X 0,Y 502.371,Z 230.335,A -85,B 0,C 180,E1 -5655.416,E2 -5655.416} C_VEL
LIN {X 0,Y 502.474,Z 226.691,A -85,B 0,C 180,E1 -5658.708,E2 -5658.708} C_VEL
LIN {X 0,Y 502.469,Z 225.899,A -85,B 0,C 180,E1 -5659.524,E2 -5659.524} C_VEL
LIN {X 0,Y 502.92,Z 225.84,A -85,B 0,C 180,E1 -5662.813,E2 -5662.813} C_VEL
LIN {X 0,Y 502.865,Z 225.848,A -85,B 0,C 180,E1 -5665.19,E2 -5665.19} C_VEL
LIN {X 0,Y 503.009,Z 225.829,A -85,B 0,C 180,E1 -5667.598,E2 -5667.598} C_VEL
LIN {X 0,Y 503.01,Z 225.828,A -85,B 0,C 180,E1 -5670,E2 -5670} C_VEL
LIN {X 0,Y 503.011,Z 225.828,A -85,B 0,C 180,E1 -5672.403,E2 -5672.403} C_VEL
LIN {X 0,Y 502.934,Z 225.839,A -85,B 0,C 180,E1 -5675.614,E2 -5675.614} C_VEL
LIN {X 0,Y 502.887,Z 225.844,A -85,B 0,C 180,E1 -5678.034,E2 -5678.034} C_VEL
LIN {X 0,Y 502.88,Z 225.848,A -85,B 0,C 180,E1 -5681.284,E2 -5681.284} C_VEL
LIN {X 0,Y 502.83,Z 225.851,A -85,B 0,C 180,E1 -5684.572,E2 -5684.572} C_VEL
LIN {X 0,Y 502.847,Z 225.848,A -85,B 0,C 180,E1 -5687.908,E2 -5687.908} C_VEL
LIN {X 0,Y 502.816,Z 225.853,A -85,B 0,C 180,E1 -5690.538,E2 -5690.538} C_VEL
LIN {X 0,Y 502.801,Z 225.857,A -85,B 0,C 180,E1 -5693.04,E2 -5693.04} C_VEL
LIN {X 0,Y 502.83,Z 225.852,A -85,B 0,C 180,E1 -5695.676,E2 -5695.676} C_VEL
LIN {X 0,Y 502.827,Z 225.853,A -85,B 0,C 180,E1 -5698.374,E2 -5698.374} C_VEL
LIN {X 0,Y 502.784,Z 225.858,A -85,B 0,C 180,E1 -5701.501,E2 -5701.501} C_VEL
LIN {X 0,Y 502.795,Z 225.856,A -85,B 0,C 180,E1 -5704.446,E2 -5704.446} C_VEL
LIN {X 0,Y 502.769,Z 225.86,A -85,B 0,C 180,E1 -5707.18,E2 -5707.18} C_VEL
LIN {X 0,Y 502.816,Z 225.854,A -85,B 0,C 180,E1 -5710.013,E2 -5710.013} C_VEL
LIN {X 0,Y 502.816,Z 225.854,A -85,B 0,C 180,E1 -5712.204,E2 -5712.204} C_VEL
LIN {X 0,Y 502.791,Z 225.855,A -85,B 0,C 180,E1 -5715.47,E2 -5715.47} C_VEL
LIN {X 0,Y 502.821,Z 225.852,A -85,B 0,C 180,E1 -5717.866,E2 -5717.866} C_VEL
LIN {X 0,Y 502.814,Z 225.853,A -85,B 0,C 180,E1 -5721.028,E2 -5721.028} C_VEL
LIN {X 0,Y 502.778,Z 225.86,A -85,B 0,C 180,E1 -5724.169,E2 -5724.169} C_VEL
LIN {X 0,Y 502.827,Z 225.851,A -85,B 0,C 180,E1 -5726.995,E2 -5726.995} C_VEL
LIN {X 0,Y 502.826,Z 225.853,A -85,B 0,C 180,E1 -5730.063,E2 -5730.063} C_VEL
LIN {X 0,Y 502.83,Z 225.854,A -85,B 0,C 180,E1 -5732.535,E2 -5732.535} C_VEL
LIN {X 0,Y 502.825,Z 225.852,A -85,B 0,C 180,E1 -5735.3,E2 -5735.3} C_VEL
LIN {X 0,Y 502.791,Z 225.857,A -85,B 0,C 180,E1 -5737.829,E2 -5737.829} C_VEL
LIN {X 0,Y 502.824,Z 225.853,A -85,B 0,C 180,E1 -5740.402,E2 -5740.402} C_VEL
LIN {X 0,Y 502.835,Z 225.851,A -85,B 0,C 180,E1 -5742.933,E2 -5742.933} C_VEL
LIN {X 0,Y 502.844,Z 225.849,A -85,B 0,C 180,E1 -5745.431,E2 -5745.431} C_VEL
LIN {X 0,Y 502.877,Z 225.845,A -85,B 0,C 180,E1 -5748.718,E2 -5748.718} C_VEL
LIN {X 0,Y 502.88,Z 225.846,A -85,B 0,C 180,E1 -5751.968,E2 -5751.968} C_VEL
LIN {X 0,Y 502.939,Z 225.838,A -85,B 0,C 180,E1 -5754.388,E2 -5754.388} C_VEL
LIN {X 0,Y 503.024,Z 225.829,A -85,B 0,C 180,E1 -5757.599,E2 -5757.599} C_VEL
LIN {X 0,Y 503.03,Z 225.829,A -85,B 0,C 180,E1 -5760.001,E2 -5760.001} C_VEL
LIN {X 0,Y 503.025,Z 225.828,A -85,B 0,C 180,E1 -5762.404,E2 -5762.404} C_VEL
LIN {X 0,Y 502.931,Z 225.84,A -85,B 0,C 180,E1 -5765.615,E2 -5765.615} C_VEL
LIN {X 0,Y 502.868,Z 225.846,A -85,B 0,C 180,E1 -5768.845,E2 -5768.845} C_VEL
LIN {X 0,Y 502.85,Z 225.849,A -85,B 0,C 180,E1 -5772.103,E2 -5772.103} C_VEL
LIN {X 0,Y 502.854,Z 225.85,A -85,B 0,C 180,E1 -5775.401,E2 -5775.401} C_VEL
LIN {X 0,Y 502.852,Z 225.848,A -85,B 0,C 180,E1 -5778.123,E2 -5778.123} C_VEL
LIN {X 0,Y 502.835,Z 225.852,A -85,B 0,C 180,E1 -5780.537,E2 -5780.537} C_VEL
LIN {X 0,Y 502.793,Z 225.857,A -85,B 0,C 180,E1 -5783.042,E2 -5783.042} C_VEL
LIN {X 0,Y 502.851,Z 225.85,A -85,B 0,C 180,E1 -5786.557,E2 -5786.557} C_VEL
LIN {X 0,Y 502.829,Z 225.852,A -85,B 0,C 180,E1 -5789.289,E2 -5789.289} C_VEL
LIN {X 0,Y 502.788,Z 225.858,A -85,B 0,C 180,E1 -5792.085,E2 -5792.085} C_VEL
LIN {X 0,Y 502.801,Z 225.856,A -85,B 0,C 180,E1 -5794.967,E2 -5794.967} C_VEL
LIN {X 0,Y 502.799,Z 225.857,A -85,B 0,C 180,E1 -5797.954,E2 -5797.954} C_VEL
LIN {X 0,Y 502.826,Z 225.852,A -85,B 0,C 180,E1 -5801.066,E2 -5801.066} C_VEL
LIN {X 0,Y 502.792,Z 225.855,A -85,B 0,C 180,E1 -5804.53,E2 -5804.53} C_VEL
LIN {X 0,Y 502.801,Z 225.857,A -85,B 0,C 180,E1 -5807.861,E2 -5807.861} C_VEL
LIN {X 0,Y 502.811,Z 225.913,A -85,B 0,C 180,E1 -5810.572,E2 -5810.572} C_VEL
LIN {X 0,Y 503.943,Z 232.149,A -85,B 0,C 180,E1 -5813.153,E2 -5813.153} C_VEL
LIN {X 0,Y 504.256,Z 236,A -85,B 0,C 180,E1 -5814.662,E2 -5814.662} C_VEL
LIN {X 0,Y 503.954,Z 244.063,A -85,B 0,C 180,E1 -5817.526,E2 -5817.526} C_VEL
LIN {X 0,Y 503.658,Z 252.158,A -85,B 0,C 180,E1 -5820.326,E2 -5820.326} C_VEL
LIN {X 0,Y 503.444,Z 259.964,A -85,B 0,C 180,E1 -5822.988,E2 -5822.988} C_VEL
LIN {X 0,Y 503.215,Z 268.214,A -85,B 0,C 180,E1 -5825.669,E2 -5825.669} C_VEL
LIN {X 0,Y 502.97,Z 277.519,A -85,B 0,C 180,E1 -5828.697,E2 -5828.697} C_VEL
LIN {X 0,Y 502.719,Z 287.597,A -85,B 0,C 180,E1 -5831.924,E2 -5831.924} C_VEL
LIN {X 0,Y 502.516,Z 297.692,A -85,B 0,C 180,E1 -5835.103,E2 -5835.103} C_VEL
LIN {X 0,Y 502.487,Z 299.581,A -85,B 0,C 180,E1 -5835.693,E2 -5835.693} C_VEL
LIN {X 0,Y 504.674,Z 313.082,A -85,B 0,C 180,E1 -5836.074,E2 -5836.074} C_VEL
LIN {X 0,Y 504.396,Z 326.103,A -85,B 0,C 180,E1 -5836.554,E2 -5836.554} C_VEL
LIN {X 0,Y 504.034,Z 338.52,A -85,B 0,C 180,E1 -5837.187,E2 -5837.187} C_VEL
LIN {X 0,Y 503.699,Z 349.583,A -85,B 0,C 180,E1 -5837.919,E2 -5837.919} C_VEL
LIN {X 0,Y 503.367,Z 360.465,A -85,B 0,C 180,E1 -5838.83,E2 -5838.83} C_VEL
LIN {X 0,Y 503.024,Z 369.33,A -85,B 0,C 180,E1 -5839.738,E2 -5839.738} C_VEL
LIN {X 0,Y 502.706,Z 378.958,A -85,B 0,C 180,E1 -5840.951,E2 -5840.951} C_VEL
LIN {X 0,Y 502.472,Z 386.619,A -85,B 0,C 180,E1 -5842.162,E2 -5842.162} C_VEL
LIN {X 0,Y 502.258,Z 393.678,A -85,B 0,C 180,E1 -5843.572,E2 -5843.572} C_VEL
LIN {X 0,Y 502.186,Z 398.371,A -85,B 0,C 180,E1 -5844.78,E2 -5844.78} C_VEL
LIN {X 0,Y 502.152,Z 401.957,A -85,B 0,C 180,E1 -5845.987,E2 -5845.987} C_VEL
LIN {X 0,Y 502.122,Z 403.807,A -85,B 0,C 180,E1 -5846.79,E2 -5846.79} C_VEL
LIN {X 0,Y 502.067,Z 405.195,A -85,B 0,C 180,E1 -5847.593,E2 -5847.593} C_VEL
LIN {X 0,Y 501.991,Z 406.785,A -85,B 0,C 180,E1 -5849.197,E2 -5849.197} C_VEL
LIN {X 0,Y 501.98,Z 407,A -85,B 0,C 180,E1 -5850,E2 -5850} C_VEL
LIN {X 0,Y 502.036,Z 406.185,A -85,B 0,C 180,E1 -5851.604,E2 -5851.604} C_VEL
LIN {X 0,Y 502.067,Z 405.198,A -85,B 0,C 180,E1 -5852.406,E2 -5852.406} C_VEL
LIN {X 0,Y 502.121,Z 403.811,A -85,B 0,C 180,E1 -5853.209,E2 -5853.209} C_VEL
LIN {X 0,Y 502.129,Z 400.897,A -85,B 0,C 180,E1 -5854.415,E2 -5854.415} C_VEL
LIN {X 0,Y 502.26,Z 396.95,A -85,B 0,C 180,E1 -5855.621,E2 -5855.621} C_VEL
LIN {X 0,Y 502.336,Z 390.979,A -85,B 0,C 180,E1 -5857.011,E2 -5857.011} C_VEL
LIN {X 0,Y 502.543,Z 384.239,A -85,B 0,C 180,E1 -5858.241,E2 -5858.241} C_VEL
LIN {X 0,Y 502.812,Z 375.995,A -85,B 0,C 180,E1 -5859.452,E2 -5859.452} C_VEL
LIN {X 0,Y 503.074,Z 367.544,A -85,B 0,C 180,E1 -5860.463,E2 -5860.463} C_VEL
LIN {X 0,Y 503.491,Z 357.1,A -85,B 0,C 180,E1 -5861.473,E2 -5861.473} C_VEL
LIN {X 0,Y 503.796,Z 345.426,A -85,B 0,C 180,E1 -5862.378,E2 -5862.378} C_VEL
LIN {X 0,Y 504.172,Z 333.499,A -85,B 0,C 180,E1 -5863.092,E2 -5863.092} C_VEL
LIN {X 0,Y 504.518,Z 321.18,A -85,B 0,C 180,E1 -5863.647,E2 -5863.647} C_VEL
LIN {X 0,Y 504.538,Z 312.193,A -85,B 0,C 180,E1 -5863.954,E2 -5863.954} C_VEL
LIN {X 0,Y 502.468,Z 299.532,A -85,B 0,C 180,E1 -5864.323,E2 -5864.323} C_VEL
LIN {X 0,Y 502.664,Z 289.437,A -85,B 0,C 180,E1 -5867.493,E2 -5867.493} C_VEL
LIN {X 0,Y 502.905,Z 279.832,A -85,B 0,C 180,E1 -5870.557,E2 -5870.557} C_VEL
LIN {X 0,Y 503.139,Z 270.903,A -85,B 0,C 180,E1 -5873.459,E2 -5873.459} C_VEL
LIN {X 0,Y 503.394,Z 260.854,A -85,B 0,C 180,E1 -5876.68,E2 -5876.68} C_VEL
LIN {X 0,Y 503.579,Z 253.239,A -85,B 0,C 180,E1 -5879.239,E2 -5879.239} C_VEL
LIN {X 0,Y 503.866,Z 245.151,A -85,B 0,C 180,E1 -5882.007,E2 -5882.007} C_VEL
LIN {X 0,Y 504.217,Z 237.131,A -85,B 0,C 180,E1 -5884.852,E2 -5884.852} C_VEL
LIN {X 0,Y 504.11,Z 233.106,A -85,B 0,C 180,E1 -5886.399,E2 -5886.399} C_VEL
LIN {X 0,Y 502.791,Z 225.858,A -85,B 0,C 180,E1 -5889.493,E2 -5889.493} C_VEL
LIN {X 0,Y 502.804,Z 225.859,A -85,B 0,C 180,E1 -5892.198,E2 -5892.198} C_VEL
LIN {X 0,Y 502.802,Z 225.857,A -85,B 0,C 180,E1 -5895.467,E2 -5895.467} C_VEL
LIN {X 0,Y 502.828,Z 225.853,A -85,B 0,C 180,E1 -5899.003,E2 -5899.003} C_VEL
LIN {X 0,Y 502.795,Z 225.858,A -85,B 0,C 180,E1 -5902.045,E2 -5902.045} C_VEL
LIN {X 0,Y 502.799,Z 225.857,A -85,B 0,C 180,E1 -5905.033,E2 -5905.033} C_VEL
LIN {X 0,Y 502.783,Z 225.86,A -85,B 0,C 180,E1 -5907.914,E2 -5907.914} C_VEL
LIN {X 0,Y 502.824,Z 225.852,A -85,B 0,C 180,E1 -5910.711,E2 -5910.711} C_VEL
LIN {X 0,Y 502.881,Z 225.847,A -85,B 0,C 180,E1 -5913.434,E2 -5913.434} C_VEL
LIN {X 0,Y 502.791,Z 225.857,A -85,B 0,C 180,E1 -5916.085,E2 -5916.085} C_VEL
LIN {X 0,Y 502.783,Z 225.858,A -85,B 0,C 180,E1 -5918.688,E2 -5918.688} C_VEL
LIN {X 0,Y 502.829,Z 225.852,A -85,B 0,C 180,E1 -5921.247,E2 -5921.247} C_VEL
LIN {X 0,Y 502.821,Z 225.854,A -85,B 0,C 180,E1 -5923.766,E2 -5923.766} C_VEL
LIN {X 0,Y 502.829,Z 225.852,A -85,B 0,C 180,E1 -5926.253,E2 -5926.253} C_VEL
LIN {X 0,Y 502.875,Z 225.848,A -85,B 0,C 180,E1 -5928.716,E2 -5928.716} C_VEL
LIN {X 0,Y 502.899,Z 225.844,A -85,B 0,C 180,E1 -5931.965,E2 -5931.965} C_VEL
LIN {X 0,Y 502.937,Z 225.839,A -85,B 0,C 180,E1 -5934.385,E2 -5934.385} C_VEL
LIN {X 0,Y 503.021,Z 225.827,A -85,B 0,C 180,E1 -5937.596,E2 -5937.596} C_VEL
LIN {X 0,Y 503.022,Z 225.828,A -85,B 0,C 180,E1 -5939.999,E2 -5939.999} C_VEL
LIN {X 0,Y 503.019,Z 225.83,A -85,B 0,C 180,E1 -5942.401,E2 -5942.401} C_VEL
LIN {X 0,Y 502.933,Z 225.841,A -85,B 0,C 180,E1 -5945.612,E2 -5945.612} C_VEL
LIN {X 0,Y 502.897,Z 225.844,A -85,B 0,C 180,E1 -5948.032,E2 -5948.032} C_VEL
LIN {X 0,Y 502.825,Z 225.855,A -85,B 0,C 180,E1 -5951.283,E2 -5951.283} C_VEL
LIN {X 0,Y 502.542,Z 226.054,A -85,B 0,C 180,E1 -5953.752,E2 -5953.752} C_VEL
LIN {X 0,Y 502.503,Z 228.749,A -85,B 0,C 180,E1 -5956.242,E2 -5956.242} C_VEL
LIN {X 0,Y 502.469,Z 231.481,A -85,B 0,C 180,E1 -5958.764,E2 -5958.764} C_VEL
LIN {X 0,Y 502.374,Z 234.236,A -85,B 0,C 180,E1 -5961.328,E2 -5961.328} C_VEL
LIN {X 0,Y 502.329,Z 237.069,A -85,B 0,C 180,E1 -5963.935,E2 -5963.935} C_VEL
LIN {X 0,Y 502.303,Z 239.979,A -85,B 0,C 180,E1 -5966.596,E2 -5966.596} C_VEL
LIN {X 0,Y 502.237,Z 243.494,A -85,B 0,C 180,E1 -5969.822,E2 -5969.822} C_VEL
LIN {X 0,Y 502.223,Z 246.876,A -85,B 0,C 180,E1 -5972.832,E2 -5972.832} C_VEL
LIN {X 0,Y 504.695,Z 258.253,A -85,B 0,C 180,E1 -5973.216,E2 -5973.216} C_VEL
LIN {X 0,Y 504.495,Z 271.252,A -85,B 0,C 180,E1 -5973.73,E2 -5973.73} C_VEL
LIN {X 0,Y 504.123,Z 283.261,A -85,B 0,C 180,E1 -5974.373,E2 -5974.373} C_VEL
LIN {X 0,Y 503.78,Z 294.137,A -85,B 0,C 180,E1 -5975.13,E2 -5975.13} C_VEL
LIN {X 0,Y 503.472,Z 304.222,A -85,B 0,C 180,E1 -5976.002,E2 -5976.002} C_VEL
LIN {X 0,Y 503.132,Z 314.221,A -85,B 0,C 180,E1 -5977.069,E2 -5977.069} C_VEL
LIN {X 0,Y 502.834,Z 322.797,A -85,B 0,C 180,E1 -5978.212,E2 -5978.212} C_VEL
LIN {X 0,Y 502.583,Z 329.752,A -85,B 0,C 180,E1 -5979.351,E2 -5979.351} C_VEL
LIN {X 0,Y 502.379,Z 335.405,A -85,B 0,C 180,E1 -5980.492,E2 -5980.492} C_VEL
LIN {X 0,Y 502.32,Z 339.883,A -85,B 0,C 180,E1 -5981.617,E2 -5981.617} C_VEL
LIN {X 0,Y 502.238,Z 343.396,A -85,B 0,C 180,E1 -5982.738,E2 -5982.738} C_VEL
LIN {X 0,Y 502.137,Z 346.024,A -85,B 0,C 180,E1 -5983.85,E2 -5983.85} C_VEL
LIN {X 0,Y 502.112,Z 347.096,A -85,B 0,C 180,E1 -5984.453,E2 -5984.453} C_VEL
LIN {X 0,Y 502.059,Z 348.47,A -85,B 0,C 180,E1 -5985.581,E2 -5985.581} C_VEL
LIN {X 0,Y 502.042,Z 349.072,A -85,B 0,C 180,E1 -5986.711,E2 -5986.711} C_VEL
LIN {X 0,Y 502.019,Z 348.688,A -85,B 0,C 180,E1 -5988.129,E2 -5988.129} C_VEL
LIN {X 0,Y 502.062,Z 347.8,A -85,B 0,C 180,E1 -5989.102,E2 -5989.102} C_VEL
LIN {X 0,Y 502.114,Z 345.755,A -85,B 0,C 180,E1 -5990.335,E2 -5990.335} C_VEL
LIN {X 0,Y 502.219,Z 342.739,A -85,B 0,C 180,E1 -5991.553,E2 -5991.553} C_VEL
LIN {X 0,Y 501.609,Z 340.908,A -85,B 0,C 180,E1 -5992.191,E2 -5992.191} C_VEL
LIN {X 0,Y 498.822,Z 337.461,A -85,B 0,C 180,E1 -5993.209,E2 -5993.209} C_VEL
LIN {X 0,Y 496.076,Z 333.282,A -85,B 0,C 180,E1 -5994.2,E2 -5994.2} C_VEL
LIN {X 0,Y 495.539,Z 330.302,A -85,B 0,C 180,E1 -5994.789,E2 -5994.789} C_VEL
LIN {X 0,Y 495.795,Z 323.34,A -85,B 0,C 180,E1 -5995.95,E2 -5995.95} C_VEL
LIN {X 0,Y 496.074,Z 315.992,A -85,B 0,C 180,E1 -5996.96,E2 -5996.96} C_VEL
LIN {X 0,Y 496.427,Z 306.53,A -85,B 0,C 180,E1 -5998.031,E2 -5998.031} C_VEL
LIN {X 0,Y 496.763,Z 296.953,A -85,B 0,C 180,E1 -5998.91,E2 -5998.91} C_VEL
LIN {X 0,Y 497.135,Z 285.094,A -85,B 0,C 180,E1 -5999.78,E2 -5999.78} C_VEL
LIN {X 0,Y 497.518,Z 272.654,A -85,B 0,C 180,E1 -6000.486,E2 -6000.486} C_VEL
LIN {X 0,Y 497.809,Z 259.497,A -85,B 0,C 180,E1 -6001.026,E2 -6001.026} C_VEL
LIN {X 0,Y 495.468,Z 248.418,A -85,B 0,C 180,E1 -6001.418,E2 -6001.418} C_VEL
LIN {X 0,Y 495.123,Z 246.663,A -85,B 0,C 180,E1 -6001.477,E2 -6001.477} C_VEL
LIN {X 0,Y 495.151,Z 243.899,A -85,B 0,C 180,E1 -6003.897,E2 -6003.897} C_VEL
LIN {X 0,Y 495.156,Z 240.854,A -85,B 0,C 180,E1 -6006.584,E2 -6006.584} C_VEL
LIN {X 0,Y 495.174,Z 237.578,A -85,B 0,C 180,E1 -6009.504,E2 -6009.504} C_VEL
LIN {X 0,Y 495.249,Z 234.061,A -85,B 0,C 180,E1 -6012.663,E2 -6012.663} C_VEL
LIN {X 0,Y 495.291,Z 231.255,A -85,B 0,C 180,E1 -6015.202,E2 -6015.202} C_VEL
LIN {X 0,Y 495.413,Z 227.574,A -85,B 0,C 180,E1 -6018.545,E2 -6018.545} C_VEL
LIN {X 0,Y 495.411,Z 226.779,A -85,B 0,C 180,E1 -6019.373,E2 -6019.373} C_VEL
LIN {X 0,Y 495.876,Z 226.718,A -85,B 0,C 180,E1 -6022.777,E2 -6022.777} C_VEL
LIN {X 0,Y 495.834,Z 226.724,A -85,B 0,C 180,E1 -6025.122,E2 -6025.122} C_VEL
LIN {X 0,Y 495.978,Z 226.705,A -85,B 0,C 180,E1 -6027.564,E2 -6027.564} C_VEL
LIN {X 0,Y 495.981,Z 226.704,A -85,B 0,C 180,E1 -6030,E2 -6030} C_VEL
LIN {X 0,Y 495.979,Z 226.704,A -85,B 0,C 180,E1 -6032.437,E2 -6032.437} C_VEL
LIN {X 0,Y 495.889,Z 226.716,A -85,B 0,C 180,E1 -6035.694,E2 -6035.694} C_VEL
LIN {X 0,Y 495.858,Z 226.72,A -85,B 0,C 180,E1 -6038.149,E2 -6038.149} C_VEL
LIN {X 0,Y 495.854,Z 226.721,A -85,B 0,C 180,E1 -6041.446,E2 -6041.446} C_VEL
LIN {X 0,Y 495.775,Z 226.731,A -85,B 0,C 180,E1 -6044.784,E2 -6044.784} C_VEL
LIN {X 0,Y 495.774,Z 226.732,A -85,B 0,C 180,E1 -6047.319,E2 -6047.319} C_VEL
LIN {X 0,Y 495.764,Z 226.732,A -85,B 0,C 180,E1 -6049.891,E2 -6049.891} C_VEL
LIN {X 0,Y 495.773,Z 226.731,A -85,B 0,C 180,E1 -6052.87,E2 -6052.87} C_VEL
LIN {X 0,Y 495.787,Z 226.729,A -85,B 0,C 180,E1 -6056.068,E2 -6056.068} C_VEL
LIN {X 0,Y 495.759,Z 226.733,A -85,B 0,C 180,E1 -6058.816,E2 -6058.816} C_VEL
LIN {X 0,Y 495.746,Z 226.734,A -85,B 0,C 180,E1 -6061.727,E2 -6061.727} C_VEL
LIN {X 0,Y 495.765,Z 226.732,A -85,B 0,C 180,E1 -6064.697,E2 -6064.697} C_VEL
LIN {X 0,Y 495.721,Z 226.737,A -85,B 0,C 180,E1 -6067.563,E2 -6067.563} C_VEL
LIN {X 0,Y 495.783,Z 226.731,A -85,B 0,C 180,E1 -6070.053,E2 -6070.053} C_VEL
LIN {X 0,Y 495.754,Z 226.733,A -85,B 0,C 180,E1 -6072.88,E2 -6072.88} C_VEL
LIN {X 0,Y 495.727,Z 226.738,A -85,B 0,C 180,E1 -6076.001,E2 -6076.001} C_VEL
LIN {X 0,Y 495.76,Z 226.733,A -85,B 0,C 180,E1 -6078.707,E2 -6078.707} C_VEL
LIN {X 0,Y 495.756,Z 226.731,A -85,B 0,C 180,E1 -6081.411,E2 -6081.411} C_VEL
LIN {X 0,Y 495.75,Z 226.735,A -85,B 0,C 180,E1 -6084.465,E2 -6084.465} C_VEL
LIN {X 0,Y 495.764,Z 226.73,A -85,B 0,C 180,E1 -6087.408,E2 -6087.408} C_VEL
LIN {X 0,Y 495.777,Z 226.733,A -85,B 0,C 180,E1 -6090.256,E2 -6090.256} C_VEL
LIN {X 0,Y 495.819,Z 226.723,A -85,B 0,C 180,E1 -6093.252,E2 -6093.252} C_VEL
LIN {X 0,Y 495.749,Z 226.733,A -85,B 0,C 180,E1 -6095.727,E2 -6095.727} C_VEL
LIN {X 0,Y 495.745,Z 226.736,A -85,B 0,C 180,E1 -6098.373,E2 -6098.373} C_VEL
LIN {X 0,Y 495.783,Z 226.73,A -85,B 0,C 180,E1 -6100.973,E2 -6100.973} C_VEL
LIN {X 0,Y 495.78,Z 226.732,A -85,B 0,C 180,E1 -6103.532,E2 -6103.532} C_VEL
LIN {X 0,Y 495.793,Z 226.729,A -85,B 0,C 180,E1 -6106.057,E2 -6106.057} C_VEL
LIN {X 0,Y 495.852,Z 226.72,A -85,B 0,C 180,E1 -6108.556,E2 -6108.556} C_VEL
LIN {X 0,Y 495.836,Z 226.724,A -85,B 0,C 180,E1 -6111.853,E2 -6111.853} C_VEL
LIN {X 0,Y 495.897,Z 226.715,A -85,B 0,C 180,E1 -6114.308,E2 -6114.308} C_VEL
LIN {X 0,Y 495.993,Z 226.705,A -85,B 0,C 180,E1 -6117.565,E2 -6117.565} C_VEL
LIN {X 0,Y 496.001,Z 226.704,A -85,B 0,C 180,E1 -6120.001,E2 -6120.001} C_VEL
LIN {X 0,Y 495.994,Z 226.703,A -85,B 0,C 180,E1 -6122.438,E2 -6122.438} C_VEL
LIN {X 0,Y 495.886,Z 226.718,A -85,B 0,C 180,E1 -6125.695,E2 -6125.695} C_VEL
LIN {X 0,Y 495.838,Z 226.722,A -85,B 0,C 180,E1 -6128.971,E2 -6128.971} C_VEL
LIN {X 0,Y 495.833,Z 226.723,A -85,B 0,C 180,E1 -6132.036,E2 -6132.036} C_VEL
LIN {X 0,Y 495.829,Z 226.726,A -85,B 0,C 180,E1 -6135.453,E2 -6135.453} C_VEL
LIN {X 0,Y 495.812,Z 226.724,A -85,B 0,C 180,E1 -6138.248,E2 -6138.248} C_VEL
LIN {X 0,Y 495.78,Z 226.73,A -85,B 0,C 180,E1 -6140.757,E2 -6140.757} C_VEL
LIN {X 0,Y 495.745,Z 226.735,A -85,B 0,C 180,E1 -6143.388,E2 -6143.388} C_VEL
LIN {X 0,Y 495.812,Z 226.726,A -85,B 0,C 180,E1 -6146.746,E2 -6146.746} C_VEL
LIN {X 0,Y 495.772,Z 226.732,A -85,B 0,C 180,E1 -6149.747,E2 -6149.747} C_VEL
LIN {X 0,Y 495.772,Z 226.731,A -85,B 0,C 180,E1 -6152.595,E2 -6152.595} C_VEL
LIN {X 0,Y 495.753,Z 226.735,A -85,B 0,C 180,E1 -6155.538,E2 -6155.538} C_VEL
LIN {X 0,Y 495.769,Z 226.731,A -85,B 0,C 180,E1 -6158.769,E2 -6158.769} C_VEL
LIN {X 0,Y 495.762,Z 226.733,A -85,B 0,C 180,E1 -6161.782,E2 -6161.782} C_VEL
LIN {X 0,Y 495.743,Z 226.734,A -85,B 0,C 180,E1 -6165.141,E2 -6165.141} C_VEL
LIN {X 0,Y 495.762,Z 226.733,A -85,B 0,C 180,E1 -6168.219,E2 -6168.219} C_VEL
LIN {X 0,Y 495.77,Z 226.743,A -85,B 0,C 180,E1 -6170.261,E2 -6170.261} C_VEL
LIN {X 0,Y 496.978,Z 233.432,A -85,B 0,C 180,E1 -6173.057,E2 -6173.057} C_VEL
LIN {X 0,Y 497.295,Z 237.252,A -85,B 0,C 180,E1 -6174.589,E2 -6174.589} C_VEL
LIN {X 0,Y 496.974,Z 245.264,A -85,B 0,C 180,E1 -6177.494,E2 -6177.494} C_VEL
LIN {X 0,Y 496.664,Z 253.296,A -85,B 0,C 180,E1 -6180.312,E2 -6180.312} C_VEL
LIN {X 0,Y 496.409,Z 261.355,A -85,B 0,C 180,E1 -6183.119,E2 -6183.119} C_VEL
LIN {X 0,Y 496.122,Z 270.693,A -85,B 0,C 180,E1 -6186.188,E2 -6186.188} C_VEL
LIN {X 0,Y 495.897,Z 280.292,A -85,B 0,C 180,E1 -6189.29,E2 -6189.29} C_VEL
LIN {X 0,Y 495.641,Z 289.434,A -85,B 0,C 180,E1 -6192.25,E2 -6192.25} C_VEL
LIN {X 0,Y 495.417,Z 299.581,A -85,B 0,C 180,E1 -6195.484,E2 -6195.484} C_VEL
LIN {X 0,Y 497.583,Z 312.626,A -85,B 0,C 180,E1 -6195.859,E2 -6195.859} C_VEL
LIN {X 0,Y 497.715,Z 318.49,A -85,B 0,C 180,E1 -6196.058,E2 -6196.058} C_VEL
LIN {X 0,Y 497.304,Z 331.497,A -85,B 0,C 180,E1 -6196.619,E2 -6196.619} C_VEL
LIN {X 0,Y 496.959,Z 342.842,A -85,B 0,C 180,E1 -6197.276,E2 -6197.276} C_VEL
LIN {X 0,Y 496.625,Z 353.481,A -85,B 0,C 180,E1 -6198.055,E2 -6198.055} C_VEL
LIN {X 0,Y 496.262,Z 363.642,A -85,B 0,C 180,E1 -6198.978,E2 -6198.978} C_VEL
LIN {X 0,Y 495.929,Z 372.783,A -85,B 0,C 180,E1 -6200.002,E2 -6200.002} C_VEL
LIN {X 0,Y 495.607,Z 381.685,A -85,B 0,C 180,E1 -6201.231,E2 -6201.231} C_VEL
LIN {X 0,Y 495.318,Z 388.846,A -85,B 0,C 180,E1 -6202.458,E2 -6202.458} C_VEL
LIN {X 0,Y 495.176,Z 394.686,A -85,B 0,C 180,E1 -6203.717,E2 -6203.717} C_VEL
LIN {X 0,Y 495.04,Z 399.676,A -85,B 0,C 180,E1 -6205.113,E2 -6205.113} C_VEL
LIN {X 0,Y 495.05,Z 401.957,A -85,B 0,C 180,E1 -6205.929,E2 -6205.929} C_VEL
LIN {X 0,Y 495.044,Z 403.806,A -85,B 0,C 180,E1 -6206.744,E2 -6206.744} C_VEL
LIN {X 0,Y 494.962,Z 406.183,A -85,B 0,C 180,E1 -6208.372,E2 -6208.372} C_VEL
LIN {X 0,Y 494.898,Z 407,A -85,B 0,C 180,E1 -6210,E2 -6210} C_VEL
LIN {X 0,Y 494.962,Z 406.185,A -85,B 0,C 180,E1 -6211.627,E2 -6211.627} C_VEL
LIN {X 0,Y 495.044,Z 403.811,A -85,B 0,C 180,E1 -6213.255,E2 -6213.255} C_VEL
LIN {X 0,Y 495.029,Z 400.897,A -85,B 0,C 180,E1 -6214.478,E2 -6214.478} C_VEL
LIN {X 0,Y 495.21,Z 395.806,A -85,B 0,C 180,E1 -6215.998,E2 -6215.998} C_VEL
LIN {X 0,Y 495.278,Z 389.871,A -85,B 0,C 180,E1 -6217.337,E2 -6217.337} C_VEL
LIN {X 0,Y 495.558,Z 383.006,A -85,B 0,C 180,E1 -6218.563,E2 -6218.563} C_VEL
LIN {X 0,Y 495.853,Z 374.417,A -85,B 0,C 180,E1 -6219.792,E2 -6219.792} C_VEL
LIN {X 0,Y 496.226,Z 365.603,A -85,B 0,C 180,E1 -6220.816,E2 -6220.816} C_VEL
LIN {X 0,Y 496.592,Z 355.926,A -85,B 0,C 180,E1 -6221.738,E2 -6221.738} C_VEL
LIN {X 0,Y 496.853,Z 345.144,A -85,B 0,C 180,E1 -6222.574,E2 -6222.574} C_VEL
LIN {X 0,Y 497.246,Z 333.498,A -85,B 0,C 180,E1 -6223.277,E2 -6223.277} C_VEL
LIN {X 0,Y 497.615,Z 321.179,A -85,B 0,C 180,E1 -6223.84,E2 -6223.84} C_VEL
LIN {X 0,Y 497.59,Z 312.65,A -85,B 0,C 180,E1 -6224.14,E2 -6224.14} C_VEL
LIN {X 0,Y 495.426,Z 299.532,A -85,B 0,C 180,E1 -6224.531,E2 -6224.531} C_VEL
LIN {X 0,Y 495.639,Z 289.437,A -85,B 0,C 180,E1 -6227.749,E2 -6227.749} C_VEL
LIN {X 0,Y 495.886,Z 280.17,A -85,B 0,C 180,E1 -6230.751,E2 -6230.751} C_VEL
LIN {X 0,Y 496.118,Z 270.639,A -85,B 0,C 180,E1 -6233.811,E2 -6233.811} C_VEL
LIN {X 0,Y 496.344,Z 262.468,A -85,B 0,C 180,E1 -6236.454,E2 -6236.454} C_VEL
LIN {X 0,Y 496.554,Z 254.32,A -85,B 0,C 180,E1 -6239.228,E2 -6239.228} C_VEL
LIN {X 0,Y 496.843,Z 246.54,A -85,B 0,C 180,E1 -6241.926,E2 -6241.926} C_VEL
LIN {X 0,Y 497.265,Z 238.264,A -85,B 0,C 180,E1 -6244.941,E2 -6244.941} C_VEL
LIN {X 0,Y 497.152,Z 234.478,A -85,B 0,C 180,E1 -6246.422,E2 -6246.422} C_VEL
LIN {X 0,Y 496.147,Z 228.806,A -85,B 0,C 180,E1 -6248.822,E2 -6248.822} C_VEL
LIN {X 0,Y 495.745,Z 226.737,A -85,B 0,C 180,E1 -6249.791,E2 -6249.791} C_VEL
LIN {X 0,Y 495.727,Z 226.738,A -85,B 0,C 180,E1 -6252.882,E2 -6252.882} C_VEL
LIN {X 0,Y 495.735,Z 226.735,A -85,B 0,C 180,E1 -6255.998,E2 -6255.998} C_VEL
LIN {X 0,Y 495.782,Z 226.731,A -85,B 0,C 180,E1 -6259.301,E2 -6259.301} C_VEL
LIN {X 0,Y 495.76,Z 226.734,A -85,B 0,C 180,E1 -6261.408,E2 -6261.408} C_VEL
LIN {X 0,Y 495.748,Z 226.735,A -85,B 0,C 180,E1 -6264.461,E2 -6264.461} C_VEL
LIN {X 0,Y 495.767,Z 226.732,A -85,B 0,C 180,E1 -6267.405,E2 -6267.405} C_VEL
LIN {X 0,Y 495.766,Z 226.733,A -85,B 0,C 180,E1 -6270.253,E2 -6270.253} C_VEL
LIN {X 0,Y 495.834,Z 226.726,A -85,B 0,C 180,E1 -6273.247,E2 -6273.247} C_VEL
LIN {X 0,Y 495.752,Z 226.733,A -85,B 0,C 180,E1 -6275.724,E2 -6275.724} C_VEL
LIN {X 0,Y 495.747,Z 226.735,A -85,B 0,C 180,E1 -6278.37,E2 -6278.37} C_VEL
LIN {X 0,Y 495.783,Z 226.73,A -85,B 0,C 180,E1 -6280.97,E2 -6280.97} C_VEL
LIN {X 0,Y 495.778,Z 226.732,A -85,B 0,C 180,E1 -6283.529,E2 -6283.529} C_VEL
LIN {X 0,Y 495.792,Z 226.729,A -85,B 0,C 180,E1 -6286.054,E2 -6286.054} C_VEL
LIN {X 0,Y 495.849,Z 226.722,A -85,B 0,C 180,E1 -6288.554,E2 -6288.554} C_VEL
LIN {X 0,Y 495.87,Z 226.719,A -85,B 0,C 180,E1 -6291.851,E2 -6291.851} C_VEL
LIN {X 0,Y 495.894,Z 226.717,A -85,B 0,C 180,E1 -6294.305,E2 -6294.305} C_VEL
LIN {X 0,Y 495.99,Z 226.703,A -85,B 0,C 180,E1 -6297.562,E2 -6297.562} C_VEL
LIN {X 0,Y 495.993,Z 226.704,A -85,B 0,C 180,E1 -6299.999,E2 -6299.999} C_VEL
LIN {X 0,Y 495.988,Z 226.706,A -85,B 0,C 180,E1 -6302.435,E2 -6302.435} C_VEL
LIN {X 0,Y 495.891,Z 226.718,A -85,B 0,C 180,E1 -6305.692,E2 -6305.692} C_VEL
LIN {X 0,Y 495.868,Z 226.72,A -85,B 0,C 180,E1 -6308.147,E2 -6308.147} C_VEL
LIN {X 0,Y 495.789,Z 226.732,A -85,B 0,C 180,E1 -6311.445,E2 -6311.445} C_VEL
LIN {X 0,Y 495.54,Z 226.764,A -85,B 0,C 180,E1 -6313.114,E2 -6313.114} C_VEL
LIN {X 0,Y 495.485,Z 227.106,A -85,B 0,C 180,E1 -6313.952,E2 -6313.952} C_VEL
LIN {X 0,Y 495.445,Z 229.818,A -85,B 0,C 180,E1 -6316.48,E2 -6316.48} C_VEL
LIN {X 0,Y 495.391,Z 232.561,A -85,B 0,C 180,E1 -6319.042,E2 -6319.042} C_VEL
LIN {X 0,Y 495.317,Z 235.305,A -85,B 0,C 180,E1 -6321.647,E2 -6321.647} C_VEL
LIN {X 0,Y 495.301,Z 238.703,A -85,B 0,C 180,E1 -6324.755,E2 -6324.755} C_VEL
LIN {X 0,Y 495.208,Z 242.129,A -85,B 0,C 180,E1 -6327.924,E2 -6327.924} C_VEL
LIN {X 0,Y 495.15,Z 245.196,A -85,B 0,C 180,E1 -6330.727,E2 -6330.727} C_VEL
LIN {X 0,Y 495.173,Z 247.273,A -85,B 0,C 180,E1 -6332.606,E2 -6332.606} C_VEL
LIN {X 0,Y 497.827,Z 259.347,A -85,B 0,C 180,E1 -6333.046,E2 -6333.046} C_VEL
LIN {X 0,Y 497.595,Z 272.043,A -85,B 0,C 180,E1 -6333.561,E2 -6333.561} C_VEL
LIN {X 0,Y 497.217,Z 283.677,A -85,B 0,C 180,E1 -6334.195,E2 -6334.195} C_VEL
LIN {X 0,Y 496.876,Z 294.348,A -85,B 0,C 180,E1 -6334.946,E2 -6334.946} C_VEL
LIN {X 0,Y 496.527,Z 304.572,A -85,B 0,C 180,E1 -6335.84,E2 -6335.84} C_VEL
LIN {X 0,Y 496.145,Z 314.286,A -85,B 0,C 180,E1 -6336.885,E2 -6336.885} C_VEL
LIN {X 0,Y 495.837,Z 323.07,A -85,B 0,C 180,E1 -6338.064,E2 -6338.064} C_VEL
LIN {X 0,Y 495.522,Z 331.136,A -85,B 0,C 180,E1 -6339.419,E2 -6339.419} C_VEL
LIN {X 0,Y 495.321,Z 337.317,A -85,B 0,C 180,E1 -6340.742,E2 -6340.742} C_VEL
LIN {X 0,Y 495.236,Z 341.324,A -85,B 0,C 180,E1 -6341.832,E2 -6341.832} C_VEL
LIN {X 0,Y 495.155,Z 344.513,A -85,B 0,C 180,E1 -6342.942,E2 -6342.942} C_VEL
LIN {X 0,Y 495.047,Z 346.937,A -85,B 0,C 180,E1 -6344.075,E2 -6344.075} C_VEL
LIN {X 0,Y 494.976,Z 348.586,A -85,B 0,C 180,E1 -6345.227,E2 -6345.227} C_VEL
LIN {X 0,Y 494.966,Z 349.441,A -85,B 0,C 180,E1 -6346.395,E2 -6346.395} C_VEL
LIN {X 0,Y 494.941,Z 349.452,A -85,B 0,C 180,E1 -6347.591,E2 -6347.591} C_VEL
LIN {X 0,Y 494.98,Z 348.1,A -85,B 0,C 180,E1 -6349.223,E2 -6349.223} C_VEL
LIN {X 0,Y 495.096,Z 345.202,A -85,B 0,C 180,E1 -6350.827,E2 -6350.827} C_VEL
LIN {X 0,Y 495.202,Z 340.734,A -85,B 0,C 180,E1 -6352.392,E2 -6352.392} C_VEL
LIN {X 0,Y 495.37,Z 335.535,A -85,B 0,C 180,E1 -6353.722,E2 -6353.722} C_VEL
LIN {X 0,Y 495.539,Z 330.302,A -85,B 0,C 180,E1 -6354.789,E2 -6354.789} C_VEL
LIN {X 0,Y 495.002,Z 327.158,A -85,B 0,C 180,E1 -6355.363,E2 -6355.363} C_VEL
LIN {X 0,Y 492.303,Z 321.771,A -85,B 0,C 180,E1 -6356.281,E2 -6356.281} C_VEL
LIN {X 0,Y 489.682,Z 315.832,A -85,B 0,C 180,E1 -6357.156,E2 -6357.156} C_VEL
LIN {X 0,Y 489.263,Z 311.768,A -85,B 0,C 180,E1 -6357.658,E2 -6357.658} C_VEL
LIN {X 0,Y 489.601,Z 302.248,A -85,B 0,C 180,E1 -6358.645,E2 -6358.645} C_VEL
LIN {X 0,Y 490.044,Z 291.551,A -85,B 0,C 180,E1 -6359.533,E2 -6359.533} C_VEL
LIN {X 0,Y 490.397,Z 279.805,A -85,B 0,C 180,E1 -6360.31,E2 -6360.31} C_VEL
LIN {X 0,Y 490.747,Z 268.75,A -85,B 0,C 180,E1 -6360.873,E2 -6360.873} C_VEL
LIN {X 0,Y 490.769,Z 259.169,A -85,B 0,C 180,E1 -6361.252,E2 -6361.252} C_VEL
LIN {X 0,Y 488.054,Z 247.046,A -85,B 0,C 180,E1 -6361.687,E2 -6361.687} C_VEL
LIN {X 0,Y 488.065,Z 243.951,A -85,B 0,C 180,E1 -6364.407,E2 -6364.407} C_VEL
LIN {X 0,Y 488.107,Z 240.871,A -85,B 0,C 180,E1 -6367.141,E2 -6367.141} C_VEL
LIN {X 0,Y 488.13,Z 237.924,A -85,B 0,C 180,E1 -6369.785,E2 -6369.785} C_VEL
LIN {X 0,Y 488.193,Z 235.015,A -85,B 0,C 180,E1 -6372.404,E2 -6372.404} C_VEL
LIN {X 0,Y 488.22,Z 232.201,A -85,B 0,C 180,E1 -6374.983,E2 -6374.983} C_VEL
LIN {X 0,Y 488.36,Z 228.463,A -85,B 0,C 180,E1 -6378.377,E2 -6378.377} C_VEL
LIN {X 0,Y 488.345,Z 227.659,A -85,B 0,C 180,E1 -6379.218,E2 -6379.218} C_VEL
LIN {X 0,Y 488.656,Z 227.619,A -85,B 0,C 180,E1 -6381.731,E2 -6381.731} C_VEL
LIN {X 0,Y 488.818,Z 227.599,A -85,B 0,C 180,E1 -6383.396,E2 -6383.396} C_VEL
LIN {X 0,Y 488.693,Z 227.613,A -85,B 0,C 180,E1 -6385.877,E2 -6385.877} C_VEL
LIN {X 0,Y 488.946,Z 227.581,A -85,B 0,C 180,E1 -6387.529,E2 -6387.529} C_VEL
LIN {X 0,Y 488.952,Z 227.579,A -85,B 0,C 180,E1 -6390,E2 -6390} C_VEL
LIN {X 0,Y 488.947,Z 227.58,A -85,B 0,C 180,E1 -6392.472,E2 -6392.472} C_VEL
LIN {X 0,Y 488.847,Z 227.592,A -85,B 0,C 180,E1 -6395.776,E2 -6395.776} C_VEL
LIN {X 0,Y 488.803,Z 227.598,A -85,B 0,C 180,E1 -6398.267,E2 -6398.267} C_VEL
LIN {X 0,Y 488.815,Z 227.597,A -85,B 0,C 180,E1 -6401.613,E2 -6401.613} C_VEL
LIN {X 0,Y 488.746,Z 227.608,A -85,B 0,C 180,E1 -6405.001,E2 -6405.001} C_VEL
LIN {X 0,Y 488.74,Z 227.607,A -85,B 0,C 180,E1 -6408.443,E2 -6408.443} C_VEL
LIN {X 0,Y 488.728,Z 227.609,A -85,B 0,C 180,E1 -6411.07,E2 -6411.07} C_VEL
LIN {X 0,Y 488.691,Z 227.611,A -85,B 0,C 180,E1 -6413.746,E2 -6413.746} C_VEL
LIN {X 0,Y 488.785,Z 227.603,A -85,B 0,C 180,E1 -6416.947,E2 -6416.947} C_VEL
LIN {X 0,Y 488.697,Z 227.613,A -85,B 0,C 180,E1 -6420.364,E2 -6420.364} C_VEL
LIN {X 0,Y 488.724,Z 227.608,A -85,B 0,C 180,E1 -6423.486,E2 -6423.486} C_VEL
LIN {X 0,Y 488.677,Z 227.616,A -85,B 0,C 180,E1 -6426.357,E2 -6426.357} C_VEL
LIN {X 0,Y 488.738,Z 227.606,A -85,B 0,C 180,E1 -6429.251,E2 -6429.251} C_VEL
LIN {X 0,Y 488.724,Z 227.61,A -85,B 0,C 180,E1 -6432.522,E2 -6432.522} C_VEL
LIN {X 0,Y 488.702,Z 227.61,A -85,B 0,C 180,E1 -6435.2,E2 -6435.2} C_VEL
LIN {X 0,Y 488.726,Z 227.608,A -85,B 0,C 180,E1 -6437.481,E2 -6437.481} C_VEL
LIN {X 0,Y 488.741,Z 227.608,A -85,B 0,C 180,E1 -6440.752,E2 -6440.752} C_VEL
LIN {X 0,Y 488.678,Z 227.614,A -85,B 0,C 180,E1 -6443.87,E2 -6443.87} C_VEL
LIN {X 0,Y 488.733,Z 227.607,A -85,B 0,C 180,E1 -6446.879,E2 -6446.879} C_VEL
LIN {X 0,Y 488.729,Z 227.608,A -85,B 0,C 180,E1 -6449.783,E2 -6449.783} C_VEL
LIN {X 0,Y 488.788,Z 227.599,A -85,B 0,C 180,E1 -6453.058,E2 -6453.058} C_VEL
LIN {X 0,Y 488.691,Z 227.615,A -85,B 0,C 180,E1 -6456.256,E2 -6456.256} C_VEL
LIN {X 0,Y 488.744,Z 227.604,A -85,B 0,C 180,E1 -6459.177,E2 -6459.177} C_VEL
LIN {X 0,Y 488.734,Z 227.608,A -85,B 0,C 180,E1 -6462.425,E2 -6462.425} C_VEL
LIN {X 0,Y 488.761,Z 227.603,A -85,B 0,C 180,E1 -6465.001,E2 -6465.001} C_VEL
LIN {X 0,Y 488.806,Z 227.598,A -85,B 0,C 180,E1 -6468.389,E2 -6468.389} C_VEL
LIN {X 0,Y 488.785,Z 227.604,A -85,B 0,C 180,E1 -6471.735,E2 -6471.735} C_VEL
LIN {X 0,Y 488.856,Z 227.593,A -85,B 0,C 180,E1 -6474.226,E2 -6474.226} C_VEL
LIN {X 0,Y 488.961,Z 227.58,A -85,B 0,C 180,E1 -6477.53,E2 -6477.53} C_VEL
LIN {X 0,Y 488.972,Z 227.58,A -85,B 0,C 180,E1 -6480.001,E2 -6480.001} C_VEL
LIN {X 0,Y 488.962,Z 227.579,A -85,B 0,C 180,E1 -6482.473,E2 -6482.473} C_VEL
LIN {X 0,Y 488.843,Z 227.596,A -85,B 0,C 180,E1 -6485.777,E2 -6485.777} C_VEL
LIN {X 0,Y 488.789,Z 227.601,A -85,B 0,C 180,E1 -6488.268,E2 -6488.268} C_VEL
LIN {X 0,Y 488.81,Z 227.599,A -85,B 0,C 180,E1 -6491.614,E2 -6491.614} C_VEL
LIN {X 0,Y 488.767,Z 227.603,A -85,B 0,C 180,E1 -6495.001,E2 -6495.001} C_VEL
LIN {X 0,Y 488.761,Z 227.602,A -85,B 0,C 180,E1 -6498.443,E2 -6498.443} C_VEL
LIN {X 0,Y 488.712,Z 227.61,A -85,B 0,C 180,E1 -6501.072,E2 -6501.072} C_VEL
LIN {X 0,Y 488.677,Z 227.616,A -85,B 0,C 180,E1 -6503.747,E2 -6503.747} C_VEL
LIN {X 0,Y 488.754,Z 227.605,A -85,B 0,C 180,E1 -6506.934,E2 -6506.934} C_VEL
LIN {X 0,Y 488.729,Z 227.609,A -85,B 0,C 180,E1 -6509.271,E2 -6509.271} C_VEL
LIN {X 0,Y 488.708,Z 227.611,A -85,B 0,C 180,E1 -6512.148,E2 -6512.148} C_VEL
LIN {X 0,Y 488.721,Z 227.61,A -85,B 0,C 180,E1 -6515.116,E2 -6515.116} C_VEL
LIN {X 0,Y 488.686,Z 227.616,A -85,B 0,C 180,E1 -6518.201,E2 -6518.201} C_VEL
LIN {X 0,Y 488.725,Z 227.609,A -85,B 0,C 180,E1 -6520.345,E2 -6520.345} C_VEL
LIN {X 0,Y 488.69,Z 227.611,A -85,B 0,C 180,E1 -6523.655,E2 -6523.655} C_VEL
LIN {X 0,Y 488.69,Z 227.613,A -85,B 0,C 180,E1 -6526.346,E2 -6526.346} C_VEL
LIN {X 0,Y 488.74,Z 227.609,A -85,B 0,C 180,E1 -6529.677,E2 -6529.677} C_VEL
LIN {X 0,Y 488.792,Z 227.905,A -85,B 0,C 180,E1 -6530.086,E2 -6530.086} C_VEL
LIN {X 0,Y 490.007,Z 234.652,A -85,B 0,C 180,E1 -6532.958,E2 -6532.958} C_VEL
LIN {X 0,Y 490.334,Z 239.225,A -85,B 0,C 180,E1 -6534.785,E2 -6534.785} C_VEL
LIN {X 0,Y 489.928,Z 247.807,A -85,B 0,C 180,E1 -6537.943,E2 -6537.943} C_VEL
LIN {X 0,Y 489.636,Z 254.429,A -85,B 0,C 180,E1 -6540.317,E2 -6540.317} C_VEL
LIN {X 0,Y 489.412,Z 261.78,A -85,B 0,C 180,E1 -6542.916,E2 -6542.916} C_VEL
LIN {X 0,Y 489.093,Z 270.412,A -85,B 0,C 180,E1 -6545.824,E2 -6545.824} C_VEL
LIN {X 0,Y 488.851,Z 280.697,A -85,B 0,C 180,E1 -6549.145,E2 -6549.145} C_VEL
LIN {X 0,Y 488.625,Z 289.612,A -85,B 0,C 180,E1 -6552.044,E2 -6552.044} C_VEL
LIN {X 0,Y 488.398,Z 299.707,A -85,B 0,C 180,E1 -6555.274,E2 -6555.274} C_VEL
LIN {X 0,Y 490.637,Z 313.082,A -85,B 0,C 180,E1 -6555.668,E2 -6555.668} C_VEL
LIN {X 0,Y 490.84,Z 317.73,A -85,B 0,C 180,E1 -6555.832,E2 -6555.832} C_VEL
LIN {X 0,Y 490.464,Z 330.503,A -85,B 0,C 180,E1 -6556.376,E2 -6556.376} C_VEL
LIN {X 0,Y 490.067,Z 341.857,A -85,B 0,C 180,E1 -6557.028,E2 -6557.028} C_VEL
LIN {X 0,Y 489.677,Z 353.481,A -85,B 0,C 180,E1 -6557.883,E2 -6557.883} C_VEL
LIN {X 0,Y 489.271,Z 363.642,A -85,B 0,C 180,E1 -6558.818,E2 -6558.818} C_VEL
LIN {X 0,Y 488.893,Z 372.783,A -85,B 0,C 180,E1 -6559.857,E2 -6559.857} C_VEL
LIN {X 0,Y 488.58,Z 381.685,A -85,B 0,C 180,E1 -6561.104,E2 -6561.104} C_VEL
LIN {X 0,Y 488.253,Z 388.846,A -85,B 0,C 180,E1 -6562.348,E2 -6562.348} C_VEL
LIN {X 0,Y 488.087,Z 395.114,A -85,B 0,C 180,E1 -6563.735,E2 -6563.735} C_VEL
LIN {X 0,Y 487.972,Z 399.675,A -85,B 0,C 180,E1 -6565.042,E2 -6565.042} C_VEL
LIN {X 0,Y 487.948,Z 401.957,A -85,B 0,C 180,E1 -6565.87,E2 -6565.87} C_VEL
LIN {X 0,Y 487.968,Z 403.806,A -85,B 0,C 180,E1 -6566.697,E2 -6566.697} C_VEL
LIN {X 0,Y 487.89,Z 406.182,A -85,B 0,C 180,E1 -6568.349,E2 -6568.349} C_VEL
LIN {X 0,Y 487.819,Z 407,A -85,B 0,C 180,E1 -6570,E2 -6570} C_VEL
LIN {X 0,Y 487.89,Z 406.185,A -85,B 0,C 180,E1 -6571.65,E2 -6571.65} C_VEL
LIN {X 0,Y 487.967,Z 403.811,A -85,B 0,C 180,E1 -6573.302,E2 -6573.302} C_VEL
LIN {X 0,Y 487.938,Z 400.897,A -85,B 0,C 180,E1 -6574.543,E2 -6574.543} C_VEL
LIN {X 0,Y 488.105,Z 396.95,A -85,B 0,C 180,E1 -6575.784,E2 -6575.784} C_VEL
LIN {X 0,Y 488.192,Z 390.878,A -85,B 0,C 180,E1 -6577.236,E2 -6577.236} C_VEL
LIN {X 0,Y 488.455,Z 384.239,A -85,B 0,C 180,E1 -6578.48,E2 -6578.48} C_VEL
LIN {X 0,Y 488.765,Z 375.995,A -85,B 0,C 180,E1 -6579.727,E2 -6579.727} C_VEL
LIN {X 0,Y 489.105,Z 367.544,A -85,B 0,C 180,E1 -6580.765,E2 -6580.765} C_VEL
LIN {X 0,Y 489.561,Z 357.098,A -85,B 0,C 180,E1 -6581.804,E2 -6581.804} C_VEL
LIN {X 0,Y 489.895,Z 345.888,A -85,B 0,C 180,E1 -6582.701,E2 -6582.701} C_VEL
LIN {X 0,Y 490.292,Z 335.414,A -85,B 0,C 180,E1 -6583.364,E2 -6583.364} C_VEL
LIN {X 0,Y 490.684,Z 323.777,A -85,B 0,C 180,E1 -6583.933,E2 -6583.933} C_VEL
LIN {X 0,Y 490.698,Z 313.536,A -85,B 0,C 180,E1 -6584.316,E2 -6584.316} C_VEL
LIN {X 0,Y 488.499,Z 300.511,A -85,B 0,C 180,E1 -6584.708,E2 -6584.708} C_VEL
LIN {X 0,Y 488.383,Z 299.532,A -85,B 0,C 180,E1 -6584.745,E2 -6584.745} C_VEL
LIN {X 0,Y 488.622,Z 289.615,A -85,B 0,C 180,E1 -6587.955,E2 -6587.955} C_VEL
LIN {X 0,Y 488.858,Z 280.016,A -85,B 0,C 180,E1 -6591.063,E2 -6591.063} C_VEL
LIN {X 0,Y 489.084,Z 270.275,A -85,B 0,C 180,E1 -6594.175,E2 -6594.175} C_VEL
LIN {X 0,Y 489.34,Z 261.614,A -85,B 0,C 180,E1 -6597.068,E2 -6597.068} C_VEL
LIN {X 0,Y 489.577,Z 254.056,A -85,B 0,C 180,E1 -6599.686,E2 -6599.686} C_VEL
LIN {X 0,Y 489.913,Z 245.991,A -85,B 0,C 180,E1 -6602.554,E2 -6602.554} C_VEL
LIN {X 0,Y 490.311,Z 238.928,A -85,B 0,C 180,E1 -6605.211,E2 -6605.211} C_VEL
LIN {X 0,Y 490.131,Z 235.507,A -85,B 0,C 180,E1 -6606.583,E2 -6606.583} C_VEL
LIN {X 0,Y 488.786,Z 227.905,A -85,B 0,C 180,E1 -6609.913,E2 -6609.913} C_VEL
LIN {X 0,Y 488.735,Z 227.609,A -85,B 0,C 180,E1 -6610.322,E2 -6610.322} C_VEL
LIN {X 0,Y 488.688,Z 227.616,A -85,B 0,C 180,E1 -6613.653,E2 -6613.653} C_VEL
LIN {X 0,Y 488.688,Z 227.614,A -85,B 0,C 180,E1 -6616.345,E2 -6616.345} C_VEL
LIN {X 0,Y 488.737,Z 227.609,A -85,B 0,C 180,E1 -6619.676,E2 -6619.676} C_VEL
LIN {X 0,Y 488.68,Z 227.616,A -85,B 0,C 180,E1 -6622.277,E2 -6622.277} C_VEL
LIN {X 0,Y 488.723,Z 227.61,A -85,B 0,C 180,E1 -6625.051,E2 -6625.051} C_VEL
LIN {X 0,Y 488.703,Z 227.614,A -85,B 0,C 180,E1 -6628.045,E2 -6628.045} C_VEL
LIN {X 0,Y 488.723,Z 227.608,A -85,B 0,C 180,E1 -6630.729,E2 -6630.729} C_VEL
LIN {X 0,Y 488.766,Z 227.604,A -85,B 0,C 180,E1 -6633.528,E2 -6633.528} C_VEL
LIN {X 0,Y 488.693,Z 227.614,A -85,B 0,C 180,E1 -6636.253,E2 -6636.253} C_VEL
LIN {X 0,Y 488.745,Z 227.606,A -85,B 0,C 180,E1 -6639.174,E2 -6639.174} C_VEL
LIN {X 0,Y 488.758,Z 227.605,A -85,B 0,C 180,E1 -6641.626,E2 -6641.626} C_VEL
LIN {X 0,Y 488.76,Z 227.605,A -85,B 0,C 180,E1 -6644.998,E2 -6644.998} C_VEL
LIN {X 0,Y 488.803,Z 227.599,A -85,B 0,C 180,E1 -6648.386,E2 -6648.386} C_VEL
LIN {X 0,Y 488.814,Z 227.597,A -85,B 0,C 180,E1 -6651.732,E2 -6651.732} C_VEL
LIN {X 0,Y 488.853,Z 227.594,A -85,B 0,C 180,E1 -6654.223,E2 -6654.223} C_VEL
LIN {X 0,Y 488.958,Z 227.579,A -85,B 0,C 180,E1 -6657.527,E2 -6657.527} C_VEL
LIN {X 0,Y 488.965,Z 227.579,A -85,B 0,C 180,E1 -6659.999,E2 -6659.999} C_VEL
LIN {X 0,Y 488.956,Z 227.581,A -85,B 0,C 180,E1 -6662.47,E2 -6662.47} C_VEL
LIN {X 0,Y 488.85,Z 227.595,A -85,B 0,C 180,E1 -6665.774,E2 -6665.774} C_VEL
LIN {X 0,Y 488.812,Z 227.599,A -85,B 0,C 180,E1 -6668.265,E2 -6668.265} C_VEL
LIN {X 0,Y 488.728,Z 227.613,A -85,B 0,C 180,E1 -6671.613,E2 -6671.613} C_VEL
LIN {X 0,Y 488.475,Z 227.644,A -85,B 0,C 180,E1 -6673.307,E2 -6673.307} C_VEL
LIN {X 0,Y 488.431,Z 228.154,A -85,B 0,C 180,E1 -6674.157,E2 -6674.157} C_VEL
LIN {X 0,Y 488.375,Z 230.893,A -85,B 0,C 180,E1 -6676.725,E2 -6676.725} C_VEL
LIN {X 0,Y 488.305,Z 233.626,A -85,B 0,C 180,E1 -6679.33,E2 -6679.33} C_VEL
LIN {X 0,Y 488.245,Z 236.464,A -85,B 0,C 180,E1 -6681.976,E2 -6681.976} C_VEL
LIN {X 0,Y 488.233,Z 239.608,A -85,B 0,C 180,E1 -6684.925,E2 -6684.925} C_VEL
LIN {X 0,Y 488.141,Z 242.323,A -85,B 0,C 180,E1 -6687.432,E2 -6687.432} C_VEL
LIN {X 0,Y 488.101,Z 245.39,A -85,B 0,C 180,E1 -6690.26,E2 -6690.26} C_VEL
LIN {X 0,Y 488.092,Z 247.731,A -85,B 0,C 180,E1 -6692.403,E2 -6692.403} C_VEL
LIN {X 0,Y 490.931,Z 260.198,A -85,B 0,C 180,E1 -6692.862,E2 -6692.862} C_VEL
LIN {X 0,Y 490.686,Z 273.152,A -85,B 0,C 180,E1 -6693.401,E2 -6693.401} C_VEL
LIN {X 0,Y 490.295,Z 284.652,A -85,B 0,C 180,E1 -6694.049,E2 -6694.049} C_VEL
LIN {X 0,Y 489.902,Z 296.211,A -85,B 0,C 180,E1 -6694.89,E2 -6694.89} C_VEL
LIN {X 0,Y 489.532,Z 306.318,A -85,B 0,C 180,E1 -6695.809,E2 -6695.809} C_VEL
LIN {X 0,Y 489.141,Z 316.251,A -85,B 0,C 180,E1 -6696.933,E2 -6696.933} C_VEL
LIN {X 0,Y 488.768,Z 325.151,A -85,B 0,C 180,E1 -6698.189,E2 -6698.189} C_VEL
LIN {X 0,Y 488.459,Z 332.665,A -85,B 0,C 180,E1 -6699.523,E2 -6699.523} C_VEL
LIN {X 0,Y 488.237,Z 338.765,A -85,B 0,C 180,E1 -6700.914,E2 -6700.914} C_VEL
LIN {X 0,Y 488.148,Z 342.591,A -85,B 0,C 180,E1 -6702.026,E2 -6702.026} C_VEL
LIN {X 0,Y 488.064,Z 345.725,A -85,B 0,C 180,E1 -6703.204,E2 -6703.204} C_VEL
LIN {X 0,Y 487.973,Z 347.208,A -85,B 0,C 180,E1 -6703.936,E2 -6703.936} C_VEL
LIN {X 0,Y 487.897,Z 348.929,A -85,B 0,C 180,E1 -6705.104,E2 -6705.104} C_VEL
LIN {X 0,Y 487.891,Z 349.808,A -85,B 0,C 180,E1 -6706.257,E2 -6706.257} C_VEL
LIN {X 0,Y 487.86,Z 349.926,A -85,B 0,C 180,E1 -6707.386,E2 -6707.386} C_VEL
LIN {X 0,Y 487.874,Z 349.338,A -85,B 0,C 180,E1 -6708.508,E2 -6708.508} C_VEL
LIN {X 0,Y 487.934,Z 347.807,A -85,B 0,C 180,E1 -6709.761,E2 -6709.761} C_VEL
LIN {X 0,Y 488.041,Z 345.259,A -85,B 0,C 180,E1 -6711.04,E2 -6711.04} C_VEL
LIN {X 0,Y 488.151,Z 341.537,A -85,B 0,C 180,E1 -6712.355,E2 -6712.355} C_VEL
LIN {X 0,Y 488.332,Z 335.848,A -85,B 0,C 180,E1 -6713.839,E2 -6713.839} C_VEL
LIN {X 0,Y 488.554,Z 329.752,A -85,B 0,C 180,E1 -6715.077,E2 -6715.077} C_VEL
LIN {X 0,Y 488.827,Z 322.779,A -85,B 0,C 180,E1 -6716.225,E2 -6716.225} C_VEL
LIN {X 0,Y 489.169,Z 313.97,A -85,B 0,C 180,E1 -6717.401,E2 -6717.401} C_VEL
LIN {X 0,Y 489.263,Z 311.768,A -85,B 0,C 180,E1 -6717.658,E2 -6717.658} C_VEL
LIN {X 0,Y 488.872,Z 307.544,A -85,B 0,C 180,E1 -6718.139,E2 -6718.139} C_VEL
LIN {X 0,Y 486.372,Z 300.49,A -85,B 0,C 180,E1 -6718.902,E2 -6718.902} C_VEL
LIN {X 0,Y 483.79,Z 293.008,A -85,B 0,C 180,E1 -6719.61,E2 -6719.61} C_VEL
LIN {X 0,Y 483.256,Z 288.086,A -85,B 0,C 180,E1 -6719.992,E2 -6719.992} C_VEL
LIN {X 0,Y 483.614,Z 276.966,A -85,B 0,C 180,E1 -6720.68,E2 -6720.68} C_VEL
LIN {X 0,Y 483.981,Z 264.306,A -85,B 0,C 180,E1 -6721.273,E2 -6721.273} C_VEL
LIN {X 0,Y 483.804,Z 259.881,A -85,B 0,C 180,E1 -6721.445,E2 -6721.445} C_VEL
LIN {X 0,Y 481.004,Z 247.406,A -85,B 0,C 180,E1 -6721.918,E2 -6721.918} C_VEL
LIN {X 0,Y 480.994,Z 243.987,A -85,B 0,C 180,E1 -6724.941,E2 -6724.941} C_VEL
LIN {X 0,Y 481.015,Z 240.934,A -85,B 0,C 180,E1 -6727.674,E2 -6727.674} C_VEL
LIN {X 0,Y 481.05,Z 237.941,A -85,B 0,C 180,E1 -6730.366,E2 -6730.366} C_VEL
LIN {X 0,Y 481.113,Z 235.028,A -85,B 0,C 180,E1 -6733.014,E2 -6733.014} C_VEL
LIN {X 0,Y 481.151,Z 232.192,A -85,B 0,C 180,E1 -6735.623,E2 -6735.623} C_VEL
LIN {X 0,Y 481.28,Z 229.373,A -85,B 0,C 180,E1 -6738.204,E2 -6738.204} C_VEL
LIN {X 0,Y 481.29,Z 228.538,A -85,B 0,C 180,E1 -6739.058,E2 -6739.058} C_VEL
LIN {X 0,Y 481.593,Z 228.499,A -85,B 0,C 180,E1 -6741.609,E2 -6741.609} C_VEL
LIN {X 0,Y 481.77,Z 228.476,A -85,B 0,C 180,E1 -6743.299,E2 -6743.299} C_VEL
LIN {X 0,Y 481.652,Z 228.491,A -85,B 0,C 180,E1 -6745.817,E2 -6745.817} C_VEL
LIN {X 0,Y 481.913,Z 228.457,A -85,B 0,C 180,E1 -6747.493,E2 -6747.493} C_VEL
LIN {X 0,Y 481.923,Z 228.455,A -85,B 0,C 180,E1 -6750,E2 -6750} C_VEL
LIN {X 0,Y 481.914,Z 228.456,A -85,B 0,C 180,E1 -6752.508,E2 -6752.508} C_VEL
LIN {X 0,Y 481.807,Z 228.469,A -85,B 0,C 180,E1 -6755.861,E2 -6755.861} C_VEL
LIN {X 0,Y 481.748,Z 228.477,A -85,B 0,C 180,E1 -6758.389,E2 -6758.389} C_VEL
LIN {X 0,Y 481.78,Z 228.472,A -85,B 0,C 180,E1 -6761.785,E2 -6761.785} C_VEL
LIN {X 0,Y 481.727,Z 228.481,A -85,B 0,C 180,E1 -6765.225,E2 -6765.225} C_VEL
LIN {X 0,Y 481.697,Z 228.486,A -85,B 0,C 180,E1 -6768.723,E2 -6768.723} C_VEL
LIN {X 0,Y 481.663,Z 228.488,A -85,B 0,C 180,E1 -6771.394,E2 -6771.394} C_VEL
LIN {X 0,Y 481.671,Z 228.486,A -85,B 0,C 180,E1 -6774.114,E2 -6774.114} C_VEL
LIN {X 0,Y 481.738,Z 228.479,A -85,B 0,C 180,E1 -6777.142,E2 -6777.142} C_VEL
LIN {X 0,Y 481.666,Z 228.486,A -85,B 0,C 180,E1 -6779.742,E2 -6779.742} C_VEL
LIN {X 0,Y 481.661,Z 228.49,A -85,B 0,C 180,E1 -6782.675,E2 -6782.675} C_VEL
LIN {X 0,Y 481.631,Z 228.491,A -85,B 0,C 180,E1 -6785.71,E2 -6785.71} C_VEL
LIN {X 0,Y 481.709,Z 228.481,A -85,B 0,C 180,E1 -6789.356,E2 -6789.356} C_VEL
LIN {X 0,Y 481.665,Z 228.488,A -85,B 0,C 180,E1 -6792.159,E2 -6792.159} C_VEL
LIN {X 0,Y 481.65,Z 228.491,A -85,B 0,C 180,E1 -6794.459,E2 -6794.459} C_VEL
LIN {X 0,Y 481.68,Z 228.488,A -85,B 0,C 180,E1 -6796.847,E2 -6796.847} C_VEL
LIN {X 0,Y 481.685,Z 228.486,A -85,B 0,C 180,E1 -6800.063,E2 -6800.063} C_VEL
LIN {X 0,Y 481.622,Z 228.493,A -85,B 0,C 180,E1 -6803.255,E2 -6803.255} C_VEL
LIN {X 0,Y 481.703,Z 228.484,A -85,B 0,C 180,E1 -6806.332,E2 -6806.332} C_VEL
LIN {X 0,Y 481.654,Z 228.489,A -85,B 0,C 180,E1 -6809.417,E2 -6809.417} C_VEL
LIN {X 0,Y 481.697,Z 228.485,A -85,B 0,C 180,E1 -6812.17,E2 -6812.17} C_VEL
LIN {X 0,Y 481.715,Z 228.482,A -85,B 0,C 180,E1 -6814.972,E2 -6814.972} C_VEL
LIN {X 0,Y 481.648,Z 228.491,A -85,B 0,C 180,E1 -6817.707,E2 -6817.707} C_VEL
LIN {X 0,Y 481.704,Z 228.483,A -85,B 0,C 180,E1 -6820.395,E2 -6820.395} C_VEL
LIN {X 0,Y 481.691,Z 228.484,A -85,B 0,C 180,E1 -6823.036,E2 -6823.036} C_VEL
LIN {X 0,Y 481.689,Z 228.486,A -85,B 0,C 180,E1 -6825.64,E2 -6825.64} C_VEL
LIN {X 0,Y 481.751,Z 228.478,A -85,B 0,C 180,E1 -6828.217,E2 -6828.217} C_VEL
LIN {X 0,Y 481.74,Z 228.48,A -85,B 0,C 180,E1 -6831.613,E2 -6831.613} C_VEL
LIN {X 0,Y 481.817,Z 228.47,A -85,B 0,C 180,E1 -6834.141,E2 -6834.141} C_VEL
LIN {X 0,Y 481.928,Z 228.456,A -85,B 0,C 180,E1 -6837.494,E2 -6837.494} C_VEL
LIN {X 0,Y 481.943,Z 228.455,A -85,B 0,C 180,E1 -6840.001,E2 -6840.001} C_VEL
LIN {X 0,Y 481.929,Z 228.455,A -85,B 0,C 180,E1 -6842.509,E2 -6842.509} C_VEL
LIN {X 0,Y 481.801,Z 228.473,A -85,B 0,C 180,E1 -6845.862,E2 -6845.862} C_VEL
LIN {X 0,Y 481.743,Z 228.478,A -85,B 0,C 180,E1 -6848.39,E2 -6848.39} C_VEL
LIN {X 0,Y 481.755,Z 228.479,A -85,B 0,C 180,E1 -6851.786,E2 -6851.786} C_VEL
LIN {X 0,Y 481.748,Z 228.478,A -85,B 0,C 180,E1 -6855.225,E2 -6855.225} C_VEL
LIN {X 0,Y 481.718,Z 228.48,A -85,B 0,C 180,E1 -6858.723,E2 -6858.723} C_VEL
LIN {X 0,Y 481.651,Z 228.492,A -85,B 0,C 180,E1 -6861.396,E2 -6861.396} C_VEL
LIN {X 0,Y 481.656,Z 228.488,A -85,B 0,C 180,E1 -6864.115,E2 -6864.115} C_VEL
LIN {X 0,Y 481.722,Z 228.482,A -85,B 0,C 180,E1 -6867.133,E2 -6867.133} C_VEL
LIN {X 0,Y 481.684,Z 228.487,A -85,B 0,C 180,E1 -6869.742,E2 -6869.742} C_VEL
LIN {X 0,Y 481.676,Z 228.487,A -85,B 0,C 180,E1 -6872.675,E2 -6872.675} C_VEL
LIN {X 0,Y 481.642,Z 228.492,A -85,B 0,C 180,E1 -6875.71,E2 -6875.71} C_VEL
LIN {X 0,Y 481.677,Z 228.487,A -85,B 0,C 180,E1 -6878.86,E2 -6878.86} C_VEL
LIN {X 0,Y 481.659,Z 228.489,A -85,B 0,C 180,E1 -6881.913,E2 -6881.913} C_VEL
LIN {X 0,Y 481.661,Z 228.487,A -85,B 0,C 180,E1 -6884.458,E2 -6884.458} C_VEL
LIN {X 0,Y 481.654,Z 228.49,A -85,B 0,C 180,E1 -6887.84,E2 -6887.84} C_VEL
LIN {X 0,Y 481.695,Z 228.52,A -85,B 0,C 180,E1 -6889.67,E2 -6889.67} C_VEL
LIN {X 0,Y 482.776,Z 234.575,A -85,B 0,C 180,E1 -6892.308,E2 -6892.308} C_VEL
LIN {X 0,Y 483.308,Z 238.432,A -85,B 0,C 180,E1 -6893.919,E2 -6893.919} C_VEL
LIN {X 0,Y 483.18,Z 243.804,A -85,B 0,C 180,E1 -6896.006,E2 -6896.006} C_VEL
LIN {X 0,Y 482.813,Z 252.425,A -85,B 0,C 180,E1 -6899.186,E2 -6899.186} C_VEL
LIN {X 0,Y 482.429,Z 262.2,A -85,B 0,C 180,E1 -6902.705,E2 -6902.705} C_VEL
LIN {X 0,Y 482.028,Z 271.512,A -85,B 0,C 180,E1 -6905.905,E2 -6905.905} C_VEL
LIN {X 0,Y 481.8,Z 280.955,A -85,B 0,C 180,E1 -6908.999,E2 -6908.999} C_VEL
LIN {X 0,Y 481.554,Z 290.715,A -85,B 0,C 180,E1 -6912.152,E2 -6912.152} C_VEL
LIN {X 0,Y 481.331,Z 299.707,A -85,B 0,C 180,E1 -6915.053,E2 -6915.053} C_VEL
LIN {X 0,Y 483.641,Z 313.082,A -85,B 0,C 180,E1 -6915.456,E2 -6915.456} C_VEL
LIN {X 0,Y 483.971,Z 317.729,A -85,B 0,C 180,E1 -6915.627,E2 -6915.627} C_VEL
LIN {X 0,Y 483.562,Z 330.503,A -85,B 0,C 180,E1 -6916.178,E2 -6916.178} C_VEL
LIN {X 0,Y 483.134,Z 342.18,A -85,B 0,C 180,E1 -6916.861,E2 -6916.861} C_VEL
LIN {X 0,Y 482.728,Z 353.48,A -85,B 0,C 180,E1 -6917.706,E2 -6917.706} C_VEL
LIN {X 0,Y 482.309,Z 363.642,A -85,B 0,C 180,E1 -6918.655,E2 -6918.655} C_VEL
LIN {X 0,Y 481.88,Z 372.782,A -85,B 0,C 180,E1 -6919.708,E2 -6919.708} C_VEL
LIN {X 0,Y 481.533,Z 381.685,A -85,B 0,C 180,E1 -6920.973,E2 -6920.973} C_VEL
LIN {X 0,Y 481.21,Z 388.846,A -85,B 0,C 180,E1 -6922.235,E2 -6922.235} C_VEL
LIN {X 0,Y 481.047,Z 394.373,A -85,B 0,C 180,E1 -6923.452,E2 -6923.452} C_VEL
LIN {X 0,Y 480.999,Z 398.371,A -85,B 0,C 180,E1 -6924.55,E2 -6924.55} C_VEL
LIN {X 0,Y 480.848,Z 401.957,A -85,B 0,C 180,E1 -6925.809,E2 -6925.809} C_VEL
LIN {X 0,Y 480.893,Z 403.806,A -85,B 0,C 180,E1 -6926.648,E2 -6926.648} C_VEL
LIN {X 0,Y 480.791,Z 406.182,A -85,B 0,C 180,E1 -6928.324,E2 -6928.324} C_VEL
LIN {X 0,Y 480.743,Z 407,A -85,B 0,C 180,E1 -6930,E2 -6930} C_VEL
LIN {X 0,Y 480.791,Z 406.184,A -85,B 0,C 180,E1 -6931.675,E2 -6931.675} C_VEL
LIN {X 0,Y 480.892,Z 403.811,A -85,B 0,C 180,E1 -6933.351,E2 -6933.351} C_VEL
LIN {X 0,Y 480.854,Z 400.896,A -85,B 0,C 180,E1 -6934.61,E2 -6934.61} C_VEL
LIN {X 0,Y 481.024,Z 396.95,A -85,B 0,C 180,E1 -6935.87,E2 -6935.87} C_VEL
LIN {X 0,Y 481.117,Z 390.878,A -85,B 0,C 180,E1 -6937.343,E2 -6937.343} C_VEL
LIN {X 0,Y 481.427,Z 384.238,A -85,B 0,C 180,E1 -6938.605,E2 -6938.605} C_VEL
LIN {X 0,Y 481.757,Z 375.995,A -85,B 0,C 180,E1 -6939.869,E2 -6939.869} C_VEL
LIN {X 0,Y 482.122,Z 367.544,A -85,B 0,C 180,E1 -6940.923,E2 -6940.923} C_VEL
LIN {X 0,Y 482.596,Z 357.097,A -85,B 0,C 180,E1 -6941.977,E2 -6941.977} C_VEL
LIN {X 0,Y 482.969,Z 345.885,A -85,B 0,C 180,E1 -6942.886,E2 -6942.886} C_VEL
LIN {X 0,Y 483.423,Z 333.496,A -85,B 0,C 180,E1 -6943.664,E2 -6943.664} C_VEL
LIN {X 0,Y 483.83,Z 321.177,A -85,B 0,C 180,E1 -6944.242,E2 -6944.242} C_VEL
LIN {X 0,Y 483.769,Z 314.319,A -85,B 0,C 180,E1 -6944.499,E2 -6944.499} C_VEL
LIN {X 0,Y 481.604,Z 301.142,A -85,B 0,C 180,E1 -6944.912,E2 -6944.912} C_VEL
LIN {X 0,Y 481.337,Z 299.532,A -85,B 0,C 180,E1 -6944.966,E2 -6944.966} C_VEL
LIN {X 0,Y 481.552,Z 290.711,A -85,B 0,C 180,E1 -6947.847,E2 -6947.847} C_VEL
LIN {X 0,Y 481.796,Z 280.857,A -85,B 0,C 180,E1 -6951,E2 -6951} C_VEL
LIN {X 0,Y 482.02,Z 271.306,A -85,B 0,C 180,E1 -6954.094,E2 -6954.094} C_VEL
LIN {X 0,Y 482.334,Z 261.984,A -85,B 0,C 180,E1 -6957.273,E2 -6957.273} C_VEL
LIN {X 0,Y 482.622,Z 253.792,A -85,B 0,C 180,E1 -6960.158,E2 -6960.158} C_VEL
LIN {X 0,Y 482.993,Z 245.863,A -85,B 0,C 180,E1 -6963.069,E2 -6963.069} C_VEL
LIN {X 0,Y 483.367,Z 239.382,A -85,B 0,C 180,E1 -6965.561,E2 -6965.561} C_VEL
LIN {X 0,Y 483.086,Z 236.285,A -85,B 0,C 180,E1 -6966.855,E2 -6966.855} C_VEL
LIN {X 0,Y 481.751,Z 228.868,A -85,B 0,C 180,E1 -6970.193,E2 -6970.193} C_VEL
LIN {X 0,Y 481.686,Z 228.487,A -85,B 0,C 180,E1 -6970.461,E2 -6970.461} C_VEL
LIN {X 0,Y 481.641,Z 228.494,A -85,B 0,C 180,E1 -6973.299,E2 -6973.299} C_VEL
LIN {X 0,Y 481.659,Z 228.49,A -85,B 0,C 180,E1 -6975.64,E2 -6975.64} C_VEL
LIN {X 0,Y 481.669,Z 228.489,A -85,B 0,C 180,E1 -6978.958,E2 -6978.958} C_VEL
LIN {X 0,Y 481.702,Z 228.485,A -85,B 0,C 180,E1 -6981.143,E2 -6981.143} C_VEL
LIN {X 0,Y 481.662,Z 228.49,A -85,B 0,C 180,E1 -6984.795,E2 -6984.795} C_VEL
LIN {X 0,Y 481.672,Z 228.489,A -85,B 0,C 180,E1 -6987.325,E2 -6987.325} C_VEL
LIN {X 0,Y 481.678,Z 228.487,A -85,B 0,C 180,E1 -6990.258,E2 -6990.258} C_VEL
LIN {X 0,Y 481.752,Z 228.479,A -85,B 0,C 180,E1 -6993.111,E2 -6993.111} C_VEL
LIN {X 0,Y 481.677,Z 228.486,A -85,B 0,C 180,E1 -6995.886,E2 -6995.886} C_VEL
LIN {X 0,Y 481.702,Z 228.483,A -85,B 0,C 180,E1 -6999.026,E2 -6999.026} C_VEL
LIN {X 0,Y 481.706,Z 228.481,A -85,B 0,C 180,E1 -7002.157,E2 -7002.157} C_VEL
LIN {X 0,Y 481.741,Z 228.479,A -85,B 0,C 180,E1 -7004.775,E2 -7004.775} C_VEL
LIN {X 0,Y 481.748,Z 228.478,A -85,B 0,C 180,E1 -7008.214,E2 -7008.214} C_VEL
LIN {X 0,Y 481.76,Z 228.475,A -85,B 0,C 180,E1 -7011.61,E2 -7011.61} C_VEL
LIN {X 0,Y 481.814,Z 228.471,A -85,B 0,C 180,E1 -7014.138,E2 -7014.138} C_VEL
LIN {X 0,Y 481.925,Z 228.455,A -85,B 0,C 180,E1 -7017.491,E2 -7017.491} C_VEL
LIN {X 0,Y 481.936,Z 228.455,A -85,B 0,C 180,E1 -7019.999,E2 -7019.999} C_VEL
LIN {X 0,Y 481.923,Z 228.457,A -85,B 0,C 180,E1 -7022.506,E2 -7022.506} C_VEL
LIN {X 0,Y 481.811,Z 228.471,A -85,B 0,C 180,E1 -7025.859,E2 -7025.859} C_VEL
LIN {X 0,Y 481.758,Z 228.478,A -85,B 0,C 180,E1 -7028.387,E2 -7028.387} C_VEL
LIN {X 0,Y 481.668,Z 228.492,A -85,B 0,C 180,E1 -7030.933,E2 -7030.933} C_VEL
LIN {X 0,Y 481.416,Z 228.523,A -85,B 0,C 180,E1 -7033.506,E2 -7033.506} C_VEL
LIN {X 0,Y 481.356,Z 231.056,A -85,B 0,C 180,E1 -7036.104,E2 -7036.104} C_VEL
LIN {X 0,Y 481.276,Z 233.829,A -85,B 0,C 180,E1 -7038.738,E2 -7038.738} C_VEL
LIN {X 0,Y 481.189,Z 236.618,A -85,B 0,C 180,E1 -7041.414,E2 -7041.414} C_VEL
LIN {X 0,Y 481.186,Z 239.53,A -85,B 0,C 180,E1 -7044.137,E2 -7044.137} C_VEL
LIN {X 0,Y 481.113,Z 242.582,A -85,B 0,C 180,E1 -7046.993,E2 -7046.993} C_VEL
LIN {X 0,Y 481.034,Z 245.586,A -85,B 0,C 180,E1 -7049.783,E2 -7049.783} C_VEL
LIN {X 0,Y 481.028,Z 248.302,A -85,B 0,C 180,E1 -7052.197,E2 -7052.197} C_VEL
LIN {X 0,Y 484.047,Z 261.151,A -85,B 0,C 180,E1 -7052.677,E2 -7052.677} C_VEL
LIN {X 0,Y 483.81,Z 273.273,A -85,B 0,C 180,E1 -7053.191,E2 -7053.191} C_VEL
LIN {X 0,Y 483.435,Z 284.682,A -85,B 0,C 180,E1 -7053.836,E2 -7053.836} C_VEL
LIN {X 0,Y 482.983,Z 296.468,A -85,B 0,C 180,E1 -7054.7,E2 -7054.7} C_VEL
LIN {X 0,Y 482.603,Z 306.531,A -85,B 0,C 180,E1 -7055.625,E2 -7055.625} C_VEL
LIN {X 0,Y 482.161,Z 316.111,A -85,B 0,C 180,E1 -7056.71,E2 -7056.71} C_VEL
LIN {X 0,Y 481.825,Z 323.784,A -85,B 0,C 180,E1 -7057.777,E2 -7057.777} C_VEL
LIN {X 0,Y 481.516,Z 331.459,A -85,B 0,C 180,E1 -7059.092,E2 -7059.092} C_VEL
LIN {X 0,Y 481.235,Z 337.042,A -85,B 0,C 180,E1 -7060.281,E2 -7060.281} C_VEL
LIN {X 0,Y 481.14,Z 341.481,A -85,B 0,C 180,E1 -7061.465,E2 -7061.465} C_VEL
LIN {X 0,Y 480.991,Z 345.989,A -85,B 0,C 180,E1 -7063.066,E2 -7063.066} C_VEL
LIN {X 0,Y 480.853,Z 348.691,A -85,B 0,C 180,E1 -7064.549,E2 -7064.549} C_VEL
LIN {X 0,Y 480.79,Z 349.968,A -85,B 0,C 180,E1 -7065.744,E2 -7065.744} C_VEL
LIN {X 0,Y 480.792,Z 350.412,A -85,B 0,C 180,E1 -7066.957,E2 -7066.957} C_VEL
LIN {X 0,Y 480.77,Z 350.009,A -85,B 0,C 180,E1 -7068.201,E2 -7068.201} C_VEL
LIN {X 0,Y 480.846,Z 348.71,A -85,B 0,C 180,E1 -7069.463,E2 -7069.463} C_VEL
LIN {X 0,Y 480.963,Z 345.737,A -85,B 0,C 180,E1 -7071.074,E2 -7071.074} C_VEL
LIN {X 0,Y 481.091,Z 341.108,A -85,B 0,C 180,E1 -7072.682,E2 -7072.682} C_VEL
LIN {X 0,Y 481.265,Z 336.613,A -85,B 0,C 180,E1 -7073.854,E2 -7073.854} C_VEL
LIN {X 0,Y 481.533,Z 329.559,A -85,B 0,C 180,E1 -7075.306,E2 -7075.306} C_VEL
LIN {X 0,Y 481.881,Z 321.55,A -85,B 0,C 180,E1 -7076.595,E2 -7076.595} C_VEL
LIN {X 0,Y 482.299,Z 312.357,A -85,B 0,C 180,E1 -7077.786,E2 -7077.786} C_VEL
LIN {X 0,Y 482.67,Z 302.549,A -85,B 0,C 180,E1 -7078.818,E2 -7078.818} C_VEL
LIN {X 0,Y 483.137,Z 291.32,A -85,B 0,C 180,E1 -7079.757,E2 -7079.757} C_VEL
LIN {X 0,Y 483.256,Z 288.086,A -85,B 0,C 180,E1 -7079.992,E2 -7079.992} C_VEL
LIN {X 0,Y 482.713,Z 281.301,A -85,B 0,C 180,E1 -7080.461,E2 -7080.461} C_VEL
LIN {X 0,Y 481.126,Z 274.492,A -85,B 0,C 180,E1 -7080.896,E2 -7080.896} C_VEL
LIN {X 0,Y 478.987,Z 267.594,A -85,B 0,C 180,E1 -7081.294,E2 -7081.294} C_VEL
LIN {X 0,Y 476.794,Z 260.538,A -85,B 0,C 180,E1 -7081.647,E2 -7081.647} C_VEL
LIN {X 0,Y 473.93,Z 247.805,A -85,B 0,C 180,E1 -7082.123,E2 -7082.123} C_VEL
LIN {X 0,Y 473.905,Z 244.054,A -85,B 0,C 180,E1 -7085.466,E2 -7085.466} C_VEL
LIN {X 0,Y 473.93,Z 240.961,A -85,B 0,C 180,E1 -7088.24,E2 -7088.24} C_VEL
LIN {X 0,Y 474.067,Z 237.289,A -85,B 0,C 180,E1 -7091.578,E2 -7091.578} C_VEL
LIN {X 0,Y 474.117,Z 234.082,A -85,B 0,C 180,E1 -7094.525,E2 -7094.525} C_VEL
LIN {X 0,Y 474.193,Z 230.301,A -85,B 0,C 180,E1 -7098.025,E2 -7098.025} C_VEL
LIN {X 0,Y 474.237,Z 229.417,A -85,B 0,C 180,E1 -7098.893,E2 -7098.893} C_VEL
LIN {X 0,Y 474.69,Z 229.357,A -85,B 0,C 180,E1 -7102.343,E2 -7102.343} C_VEL
LIN {X 0,Y 474.744,Z 229.352,A -85,B 0,C 180,E1 -7104.905,E2 -7104.905} C_VEL
LIN {X 0,Y 474.879,Z 229.334,A -85,B 0,C 180,E1 -7107.456,E2 -7107.456} C_VEL
LIN {X 0,Y 474.895,Z 229.33,A -85,B 0,C 180,E1 -7110,E2 -7110} C_VEL
LIN {X 0,Y 474.88,Z 229.332,A -85,B 0,C 180,E1 -7112.545,E2 -7112.545} C_VEL
LIN {X 0,Y 474.769,Z 229.346,A -85,B 0,C 180,E1 -7115.948,E2 -7115.948} C_VEL
LIN {X 0,Y 474.713,Z 229.353,A -85,B 0,C 180,E1 -7118.514,E2 -7118.514} C_VEL
LIN {X 0,Y 474.724,Z 229.351,A -85,B 0,C 180,E1 -7121.962,E2 -7121.962} C_VEL
LIN {X 0,Y 474.665,Z 229.36,A -85,B 0,C 180,E1 -7125.769,E2 -7125.769} C_VEL
LIN {X 0,Y 474.651,Z 229.362,A -85,B 0,C 180,E1 -7129.011,E2 -7129.011} C_VEL
LIN {X 0,Y 474.63,Z 229.364,A -85,B 0,C 180,E1 -7131.727,E2 -7131.727} C_VEL
LIN {X 0,Y 474.65,Z 229.363,A -85,B 0,C 180,E1 -7134.494,E2 -7134.494} C_VEL
LIN {X 0,Y 474.685,Z 229.357,A -85,B 0,C 180,E1 -7137.34,E2 -7137.34} C_VEL
LIN {X 0,Y 474.592,Z 229.37,A -85,B 0,C 180,E1 -7140.812,E2 -7140.812} C_VEL
LIN {X 0,Y 474.626,Z 229.365,A -85,B 0,C 180,E1 -7143.985,E2 -7143.985} C_VEL
LIN {X 0,Y 474.564,Z 229.373,A -85,B 0,C 180,E1 -7146.901,E2 -7146.901} C_VEL
LIN {X 0,Y 474.644,Z 229.361,A -85,B 0,C 180,E1 -7149.653,E2 -7149.653} C_VEL
LIN {X 0,Y 474.642,Z 229.363,A -85,B 0,C 180,E1 -7152.932,E2 -7152.932} C_VEL
LIN {X 0,Y 474.609,Z 229.367,A -85,B 0,C 180,E1 -7155.898,E2 -7155.898} C_VEL
LIN {X 0,Y 474.637,Z 229.364,A -85,B 0,C 180,E1 -7159.04,E2 -7159.04} C_VEL
LIN {X 0,Y 474.612,Z 229.366,A -85,B 0,C 180,E1 -7161.704,E2 -7161.704} C_VEL
LIN {X 0,Y 474.623,Z 229.365,A -85,B 0,C 180,E1 -7164.728,E2 -7164.728} C_VEL
LIN {X 0,Y 474.632,Z 229.364,A -85,B 0,C 180,E1 -7167.79,E2 -7167.79} C_VEL
LIN {X 0,Y 474.628,Z 229.364,A -85,B 0,C 180,E1 -7170.884,E2 -7170.884} C_VEL
LIN {X 0,Y 474.657,Z 229.36,A -85,B 0,C 180,E1 -7173.63,E2 -7173.63} C_VEL
LIN {X 0,Y 474.633,Z 229.364,A -85,B 0,C 180,E1 -7176.643,E2 -7176.643} C_VEL
LIN {X 0,Y 474.653,Z 229.362,A -85,B 0,C 180,E1 -7180.091,E2 -7180.091} C_VEL
LIN {X 0,Y 474.65,Z 229.361,A -85,B 0,C 180,E1 -7182.776,E2 -7182.776} C_VEL
LIN {X 0,Y 474.647,Z 229.361,A -85,B 0,C 180,E1 -7185.423,E2 -7185.423} C_VEL
LIN {X 0,Y 474.704,Z 229.357,A -85,B 0,C 180,E1 -7188.039,E2 -7188.039} C_VEL
LIN {X 0,Y 474.711,Z 229.354,A -85,B 0,C 180,E1 -7191.488,E2 -7191.488} C_VEL
LIN {X 0,Y 474.779,Z 229.348,A -85,B 0,C 180,E1 -7194.054,E2 -7194.054} C_VEL
LIN {X 0,Y 474.894,Z 229.332,A -85,B 0,C 180,E1 -7197.457,E2 -7197.457} C_VEL
LIN {X 0,Y 474.914,Z 229.331,A -85,B 0,C 180,E1 -7200.001,E2 -7200.001} C_VEL
LIN {X 0,Y 474.895,Z 229.331,A -85,B 0,C 180,E1 -7202.546,E2 -7202.546} C_VEL
LIN {X 0,Y 474.762,Z 229.349,A -85,B 0,C 180,E1 -7205.949,E2 -7205.949} C_VEL
LIN {X 0,Y 474.715,Z 229.353,A -85,B 0,C 180,E1 -7208.515,E2 -7208.515} C_VEL
LIN {X 0,Y 474.709,Z 229.355,A -85,B 0,C 180,E1 -7211.964,E2 -7211.964} C_VEL
LIN {X 0,Y 474.705,Z 229.357,A -85,B 0,C 180,E1 -7215.457,E2 -7215.457} C_VEL
LIN {X 0,Y 474.67,Z 229.36,A -85,B 0,C 180,E1 -7219.011,E2 -7219.011} C_VEL
LIN {X 0,Y 474.594,Z 229.369,A -85,B 0,C 180,E1 -7221.73,E2 -7221.73} C_VEL
LIN {X 0,Y 474.634,Z 229.362,A -85,B 0,C 180,E1 -7224.495,E2 -7224.495} C_VEL
LIN {X 0,Y 474.679,Z 229.36,A -85,B 0,C 180,E1 -7227.333,E2 -7227.333} C_VEL
LIN {X 0,Y 474.61,Z 229.365,A -85,B 0,C 180,E1 -7230.231,E2 -7230.231} C_VEL
LIN {X 0,Y 474.631,Z 229.366,A -85,B 0,C 180,E1 -7233.222,E2 -7233.222} C_VEL
LIN {X 0,Y 474.595,Z 229.367,A -85,B 0,C 180,E1 -7236.324,E2 -7236.324} C_VEL
LIN {X 0,Y 474.624,Z 229.364,A -85,B 0,C 180,E1 -7239.647,E2 -7239.647} C_VEL
LIN {X 0,Y 474.63,Z 229.363,A -85,B 0,C 180,E1 -7242.237,E2 -7242.237} C_VEL
LIN {X 0,Y 474.623,Z 229.365,A -85,B 0,C 180,E1 -7245.298,E2 -7245.298} C_VEL
LIN {X 0,Y 474.627,Z 229.366,A -85,B 0,C 180,E1 -7248.215,E2 -7248.215} C_VEL
LIN {X 0,Y 474.66,Z 229.508,A -85,B 0,C 180,E1 -7249.41,E2 -7249.41} C_VEL
LIN {X 0,Y 475.788,Z 235.775,A -85,B 0,C 180,E1 -7252.192,E2 -7252.192} C_VEL
LIN {X 0,Y 476.39,Z 240.622,A -85,B 0,C 180,E1 -7254.234,E2 -7254.234} C_VEL
LIN {X 0,Y 476.038,Z 248.54,A -85,B 0,C 180,E1 -7257.302,E2 -7257.302} C_VEL
LIN {X 0,Y 475.612,Z 256.646,A -85,B 0,C 180,E1 -7260.31,E2 -7260.31} C_VEL
LIN {X 0,Y 475.296,Z 264.586,A -85,B 0,C 180,E1 -7263.192,E2 -7263.192} C_VEL
LIN {X 0,Y 474.972,Z 272.611,A -85,B 0,C 180,E1 -7265.989,E2 -7265.989} C_VEL
LIN {X 0,Y 474.716,Z 282.238,A -85,B 0,C 180,E1 -7269.187,E2 -7269.187} C_VEL
LIN {X 0,Y 474.466,Z 291.808,A -85,B 0,C 180,E1 -7272.322,E2 -7272.322} C_VEL
LIN {X 0,Y 474.266,Z 299.599,A -85,B 0,C 180,E1 -7274.825,E2 -7274.825} C_VEL
LIN {X 0,Y 476.609,Z 313.082,A -85,B 0,C 180,E1 -7275.236,E2 -7275.236} C_VEL
LIN {X 0,Y 477.096,Z 317.729,A -85,B 0,C 180,E1 -7275.415,E2 -7275.415} C_VEL
LIN {X 0,Y 476.681,Z 330.502,A -85,B 0,C 180,E1 -7275.974,E2 -7275.974} C_VEL
LIN {X 0,Y 476.187,Z 342.671,A -85,B 0,C 180,E1 -7276.699,E2 -7276.699} C_VEL
LIN {X 0,Y 475.783,Z 353.479,A -85,B 0,C 180,E1 -7277.523,E2 -7277.523} C_VEL
LIN {X 0,Y 475.343,Z 363.642,A -85,B 0,C 180,E1 -7278.486,E2 -7278.486} C_VEL
LIN {X 0,Y 474.87,Z 372.782,A -85,B 0,C 180,E1 -7279.554,E2 -7279.554} C_VEL
LIN {X 0,Y 474.484,Z 381.685,A -85,B 0,C 180,E1 -7280.838,E2 -7280.838} C_VEL
LIN {X 0,Y 474.155,Z 388.846,A -85,B 0,C 180,E1 -7282.119,E2 -7282.119} C_VEL
LIN {X 0,Y 473.975,Z 394.739,A -85,B 0,C 180,E1 -7283.449,E2 -7283.449} C_VEL
LIN {X 0,Y 473.847,Z 399.675,A -85,B 0,C 180,E1 -7284.894,E2 -7284.894} C_VEL
LIN {X 0,Y 473.753,Z 401.957,A -85,B 0,C 180,E1 -7285.746,E2 -7285.746} C_VEL
LIN {X 0,Y 473.801,Z 403.806,A -85,B 0,C 180,E1 -7286.598,E2 -7286.598} C_VEL
LIN {X 0,Y 473.696,Z 406.181,A -85,B 0,C 180,E1 -7288.299,E2 -7288.299} C_VEL
LIN {X 0,Y 473.689,Z 406.785,A -85,B 0,C 180,E1 -7289.149,E2 -7289.149} C_VEL
LIN {X 0,Y 473.67,Z 407,A -85,B 0,C 180,E1 -7290,E2 -7290} C_VEL
LIN {X 0,Y 473.689,Z 406.786,A -85,B 0,C 180,E1 -7290.85,E2 -7290.85} C_VEL
LIN {X 0,Y 473.725,Z 405.197,A -85,B 0,C 180,E1 -7292.55,E2 -7292.55} C_VEL
LIN {X 0,Y 473.8,Z 403.811,A -85,B 0,C 180,E1 -7293.401,E2 -7293.401} C_VEL
LIN {X 0,Y 473.776,Z 400.896,A -85,B 0,C 180,E1 -7294.679,E2 -7294.679} C_VEL
LIN {X 0,Y 473.943,Z 396.95,A -85,B 0,C 180,E1 -7295.958,E2 -7295.958} C_VEL
LIN {X 0,Y 474.049,Z 390.878,A -85,B 0,C 180,E1 -7297.453,E2 -7297.453} C_VEL
LIN {X 0,Y 474.379,Z 384.238,A -85,B 0,C 180,E1 -7298.734,E2 -7298.734} C_VEL
LIN {X 0,Y 474.752,Z 375.996,A -85,B 0,C 180,E1 -7300.017,E2 -7300.017} C_VEL
LIN {X 0,Y 475.143,Z 367.544,A -85,B 0,C 180,E1 -7301.086,E2 -7301.086} C_VEL
LIN {X 0,Y 475.639,Z 357.117,A -85,B 0,C 180,E1 -7302.153,E2 -7302.153} C_VEL
LIN {X 0,Y 476.027,Z 346.047,A -85,B 0,C 180,E1 -7303.065,E2 -7303.065} C_VEL
LIN {X 0,Y 476.465,Z 335.412,A -85,B 0,C 180,E1 -7303.759,E2 -7303.759} C_VEL
LIN {X 0,Y 476.918,Z 323.777,A -85,B 0,C 180,E1 -7304.344,E2 -7304.344} C_VEL
LIN {X 0,Y 476.871,Z 315.08,A -85,B 0,C 180,E1 -7304.686,E2 -7304.686} C_VEL
LIN {X 0,Y 474.858,Z 302.749,A -85,B 0,C 180,E1 -7305.096,E2 -7305.096} C_VEL
LIN {X 0,Y 474.269,Z 299.449,A -85,B 0,C 180,E1 -7305.194,E2 -7305.194} C_VEL
LIN {X 0,Y 474.551,Z 288.916,A -85,B 0,C 180,E1 -7308.588,E2 -7308.588} C_VEL
LIN {X 0,Y 474.753,Z 279.298,A -85,B 0,C 180,E1 -7311.72,E2 -7311.72} C_VEL
LIN {X 0,Y 475.039,Z 269.61,A -85,B 0,C 180,E1 -7314.938,E2 -7314.938} C_VEL
LIN {X 0,Y 475.431,Z 260.25,A -85,B 0,C 180,E1 -7318.231,E2 -7318.231} C_VEL
LIN {X 0,Y 475.791,Z 250.91,A -85,B 0,C 180,E1 -7321.626,E2 -7321.626} C_VEL
LIN {X 0,Y 476.256,Z 243.067,A -85,B 0,C 180,E1 -7324.646,E2 -7324.646} C_VEL
LIN {X 0,Y 476.324,Z 239.303,A -85,B 0,C 180,E1 -7326.169,E2 -7326.169} C_VEL
LIN {X 0,Y 475.279,Z 233.082,A -85,B 0,C 180,E1 -7328.935,E2 -7328.935} C_VEL
LIN {X 0,Y 474.626,Z 229.367,A -85,B 0,C 180,E1 -7330.731,E2 -7330.731} C_VEL
LIN {X 0,Y 474.603,Z 229.371,A -85,B 0,C 180,E1 -7333.48,E2 -7333.48} C_VEL
LIN {X 0,Y 474.603,Z 229.369,A -85,B 0,C 180,E1 -7336.518,E2 -7336.518} C_VEL
LIN {X 0,Y 474.639,Z 229.365,A -85,B 0,C 180,E1 -7339.343,E2 -7339.343} C_VEL
LIN {X 0,Y 474.618,Z 229.367,A -85,B 0,C 180,E1 -7341.702,E2 -7341.702} C_VEL
LIN {X 0,Y 474.624,Z 229.367,A -85,B 0,C 180,E1 -7344.725,E2 -7344.725} C_VEL
LIN {X 0,Y 474.635,Z 229.365,A -85,B 0,C 180,E1 -7347.787,E2 -7347.787} C_VEL
LIN {X 0,Y 474.624,Z 229.365,A -85,B 0,C 180,E1 -7350.883,E2 -7350.883} C_VEL
LIN {X 0,Y 474.666,Z 229.36,A -85,B 0,C 180,E1 -7353.628,E2 -7353.628} C_VEL
LIN {X 0,Y 474.635,Z 229.364,A -85,B 0,C 180,E1 -7356.64,E2 -7356.64} C_VEL
LIN {X 0,Y 474.655,Z 229.359,A -85,B 0,C 180,E1 -7360.088,E2 -7360.088} C_VEL
LIN {X 0,Y 474.649,Z 229.363,A -85,B 0,C 180,E1 -7362.773,E2 -7362.773} C_VEL
LIN {X 0,Y 474.646,Z 229.363,A -85,B 0,C 180,E1 -7365.42,E2 -7365.42} C_VEL
LIN {X 0,Y 474.702,Z 229.357,A -85,B 0,C 180,E1 -7368.036,E2 -7368.036} C_VEL
LIN {X 0,Y 474.725,Z 229.351,A -85,B 0,C 180,E1 -7371.485,E2 -7371.485} C_VEL
LIN {X 0,Y 474.777,Z 229.347,A -85,B 0,C 180,E1 -7374.051,E2 -7374.051} C_VEL
LIN {X 0,Y 474.891,Z 229.331,A -85,B 0,C 180,E1 -7377.454,E2 -7377.454} C_VEL
LIN {X 0,Y 474.873,Z 229.334,A -85,B 0,C 180,E1 -7380.847,E2 -7380.847} C_VEL
LIN {X 0,Y 474.889,Z 229.333,A -85,B 0,C 180,E1 -7382.543,E2 -7382.543} C_VEL
LIN {X 0,Y 474.774,Z 229.348,A -85,B 0,C 180,E1 -7385.946,E2 -7385.946} C_VEL
LIN {X 0,Y 474.722,Z 229.355,A -85,B 0,C 180,E1 -7388.512,E2 -7388.512} C_VEL
LIN {X 0,Y 474.63,Z 229.368,A -85,B 0,C 180,E1 -7391.097,E2 -7391.097} C_VEL
LIN {X 0,Y 474.334,Z 229.412,A -85,B 0,C 180,E1 -7393.712,E2 -7393.712} C_VEL
LIN {X 0,Y 474.305,Z 232.15,A -85,B 0,C 180,E1 -7396.35,E2 -7396.35} C_VEL
LIN {X 0,Y 474.21,Z 234.93,A -85,B 0,C 180,E1 -7399.027,E2 -7399.027} C_VEL
LIN {X 0,Y 474.117,Z 237.757,A -85,B 0,C 180,E1 -7401.75,E2 -7401.75} C_VEL
LIN {X 0,Y 474.101,Z 240.714,A -85,B 0,C 180,E1 -7404.522,E2 -7404.522} C_VEL
LIN {X 0,Y 474.022,Z 243.721,A -85,B 0,C 180,E1 -7407.36,E2 -7407.36} C_VEL
LIN {X 0,Y 473.965,Z 246.828,A -85,B 0,C 180,E1 -7410.273,E2 -7410.273} C_VEL
LIN {X 0,Y 473.942,Z 248.631,A -85,B 0,C 180,E1 -7411.949,E2 -7411.949} C_VEL
LIN {X 0,Y 477.227,Z 262.771,A -85,B 0,C 180,E1 -7412.51,E2 -7412.51} C_VEL
LIN {X 0,Y 476.931,Z 274.723,A -85,B 0,C 180,E1 -7413.038,E2 -7413.038} C_VEL
LIN {X 0,Y 476.495,Z 286.054,A -85,B 0,C 180,E1 -7413.705,E2 -7413.705} C_VEL
LIN {X 0,Y 476.046,Z 297.283,A -85,B 0,C 180,E1 -7414.55,E2 -7414.55} C_VEL
LIN {X 0,Y 475.594,Z 307.949,A -85,B 0,C 180,E1 -7415.556,E2 -7415.556} C_VEL
LIN {X 0,Y 475.213,Z 316.211,A -85,B 0,C 180,E1 -7416.514,E2 -7416.514} C_VEL
LIN {X 0,Y 474.778,Z 325.383,A -85,B 0,C 180,E1 -7417.825,E2 -7417.825} C_VEL
LIN {X 0,Y 474.491,Z 332.083,A -85,B 0,C 180,E1 -7419.01,E2 -7419.01} C_VEL
LIN {X 0,Y 474.173,Z 338.48,A -85,B 0,C 180,E1 -7420.422,E2 -7420.422} C_VEL
LIN {X 0,Y 474.035,Z 343.381,A -85,B 0,C 180,E1 -7421.846,E2 -7421.846} C_VEL
LIN {X 0,Y 473.873,Z 347.219,A -85,B 0,C 180,E1 -7423.389,E2 -7423.389} C_VEL
LIN {X 0,Y 473.763,Z 349.241,A -85,B 0,C 180,E1 -7424.599,E2 -7424.599} C_VEL
LIN {X 0,Y 473.702,Z 350.438,A -85,B 0,C 180,E1 -7425.79,E2 -7425.79} C_VEL
LIN {X 0,Y 473.706,Z 350.845,A -85,B 0,C 180,E1 -7426.964,E2 -7426.964} C_VEL
LIN {X 0,Y 473.701,Z 350.496,A -85,B 0,C 180,E1 -7428.116,E2 -7428.116} C_VEL
LIN {X 0,Y 473.758,Z 349.46,A -85,B 0,C 180,E1 -7429.254,E2 -7429.254} C_VEL
LIN {X 0,Y 473.843,Z 347.572,A -85,B 0,C 180,E1 -7430.464,E2 -7430.464} C_VEL
LIN {X 0,Y 473.953,Z 344.47,A -85,B 0,C 180,E1 -7431.801,E2 -7431.801} C_VEL
LIN {X 0,Y 474.104,Z 340.101,A -85,B 0,C 180,E1 -7433.173,E2 -7433.173} C_VEL
LIN {X 0,Y 474.363,Z 333.643,A -85,B 0,C 180,E1 -7434.704,E2 -7434.704} C_VEL
LIN {X 0,Y 474.66,Z 326.627,A -85,B 0,C 180,E1 -7436.009,E2 -7436.009} C_VEL
LIN {X 0,Y 475.049,Z 318.836,A -85,B 0,C 180,E1 -7437.174,E2 -7437.174} C_VEL
LIN {X 0,Y 475.497,Z 309.122,A -85,B 0,C 180,E1 -7438.353,E2 -7438.353} C_VEL
LIN {X 0,Y 475.943,Z 298.71,A -85,B 0,C 180,E1 -7439.374,E2 -7439.374} C_VEL
LIN {X 0,Y 476.375,Z 287.761,A -85,B 0,C 180,E1 -7440.228,E2 -7440.228} C_VEL
LIN {X 0,Y 476.782,Z 275.904,A -85,B 0,C 180,E1 -7440.954,E2 -7440.954} C_VEL
LIN {X 0,Y 477.142,Z 263.669,A -85,B 0,C 180,E1 -7441.52,E2 -7441.52} C_VEL
LIN {X 0,Y 476.794,Z 260.538,A -85,B 0,C 180,E1 -7441.647,E2 -7441.647} C_VEL
LIN {X 0,Y 475.549,Z 258.452,A -85,B 0,C 180,E1 -7441.764,E2 -7441.764} C_VEL
LIN {X 0,Y 468.814,Z 253.387,A -85,B 0,C 180,E1 -7442.147,E2 -7442.147} C_VEL
LIN {X 0,Y 467.551,Z 251.251,A -85,B 0,C 180,E1 -7442.245,E2 -7442.245} C_VEL
LIN {X 0,Y 466.864,Z 248.187,A -85,B 0,C 180,E1 -7442.351,E2 -7442.351} C_VEL
LIN {X 0,Y 466.829,Z 245.141,A -85,B 0,C 180,E1 -7445.069,E2 -7445.069} C_VEL
LIN {X 0,Y 466.859,Z 242.023,A -85,B 0,C 180,E1 -7447.893,E2 -7447.893} C_VEL
LIN {X 0,Y 467.009,Z 237.97,A -85,B 0,C 180,E1 -7451.578,E2 -7451.578} C_VEL
LIN {X 0,Y 467.043,Z 234.113,A -85,B 0,C 180,E1 -7455.179,E2 -7455.179} C_VEL
LIN {X 0,Y 467.164,Z 230.298,A -85,B 0,C 180,E1 -7458.722,E2 -7458.722} C_VEL
LIN {X 0,Y 467.493,Z 230.255,A -85,B 0,C 180,E1 -7461.354,E2 -7461.354} C_VEL
LIN {X 0,Y 467.73,Z 230.223,A -85,B 0,C 180,E1 -7463.963,E2 -7463.963} C_VEL
LIN {X 0,Y 467.845,Z 230.21,A -85,B 0,C 180,E1 -7467.418,E2 -7467.418} C_VEL
LIN {X 0,Y 467.866,Z 230.206,A -85,B 0,C 180,E1 -7470,E2 -7470} C_VEL
LIN {X 0,Y 467.845,Z 230.208,A -85,B 0,C 180,E1 -7472.583,E2 -7472.583} C_VEL
LIN {X 0,Y 467.732,Z 230.222,A -85,B 0,C 180,E1 -7476.038,E2 -7476.038} C_VEL
LIN {X 0,Y 467.667,Z 230.231,A -85,B 0,C 180,E1 -7478.643,E2 -7478.643} C_VEL
LIN {X 0,Y 467.667,Z 230.23,A -85,B 0,C 180,E1 -7482.146,E2 -7482.146} C_VEL
LIN {X 0,Y 467.634,Z 230.235,A -85,B 0,C 180,E1 -7485.886,E2 -7485.886} C_VEL
LIN {X 0,Y 467.61,Z 230.24,A -85,B 0,C 180,E1 -7489.309,E2 -7489.309} C_VEL
LIN {X 0,Y 467.561,Z 230.244,A -85,B 0,C 180,E1 -7492.073,E2 -7492.073} C_VEL
LIN {X 0,Y 467.6,Z 230.241,A -85,B 0,C 180,E1 -7494.888,E2 -7494.888} C_VEL
LIN {X 0,Y 467.614,Z 230.237,A -85,B 0,C 180,E1 -7497.77,E2 -7497.77} C_VEL
LIN {X 0,Y 467.556,Z 230.246,A -85,B 0,C 180,E1 -7501.047,E2 -7501.047} C_VEL
LIN {X 0,Y 467.578,Z 230.244,A -85,B 0,C 180,E1 -7504.244,E2 -7504.244} C_VEL
LIN {X 0,Y 467.54,Z 230.248,A -85,B 0,C 180,E1 -7507.188,E2 -7507.188} C_VEL
LIN {X 0,Y 467.587,Z 230.243,A -85,B 0,C 180,E1 -7510.264,E2 -7510.264} C_VEL
LIN {X 0,Y 467.609,Z 230.24,A -85,B 0,C 180,E1 -7512.573,E2 -7512.573} C_VEL
LIN {X 0,Y 467.566,Z 230.246,A -85,B 0,C 180,E1 -7516.178,E2 -7516.178} C_VEL
LIN {X 0,Y 467.581,Z 230.243,A -85,B 0,C 180,E1 -7518.723,E2 -7518.723} C_VEL
LIN {X 0,Y 467.57,Z 230.242,A -85,B 0,C 180,E1 -7521.408,E2 -7521.408} C_VEL
LIN {X 0,Y 467.556,Z 230.248,A -85,B 0,C 180,E1 -7524.262,E2 -7524.262} C_VEL
LIN {X 0,Y 467.577,Z 230.241,A -85,B 0,C 180,E1 -7527.322,E2 -7527.322} C_VEL
LIN {X 0,Y 467.574,Z 230.243,A -85,B 0,C 180,E1 -7530.667,E2 -7530.667} C_VEL
LIN {X 0,Y 467.612,Z 230.236,A -85,B 0,C 180,E1 -7533.201,E2 -7533.201} C_VEL
LIN {X 0,Y 467.59,Z 230.241,A -85,B 0,C 180,E1 -7536.47,E2 -7536.47} C_VEL
LIN {X 0,Y 467.621,Z 230.239,A -85,B 0,C 180,E1 -7539.779,E2 -7539.779} C_VEL
LIN {X 0,Y 467.608,Z 230.239,A -85,B 0,C 180,E1 -7542.509,E2 -7542.509} C_VEL
LIN {X 0,Y 467.605,Z 230.237,A -85,B 0,C 180,E1 -7545.198,E2 -7545.198} C_VEL
LIN {X 0,Y 467.656,Z 230.234,A -85,B 0,C 180,E1 -7547.856,E2 -7547.856} C_VEL
LIN {X 0,Y 467.669,Z 230.23,A -85,B 0,C 180,E1 -7551.359,E2 -7551.359} C_VEL
LIN {X 0,Y 467.743,Z 230.224,A -85,B 0,C 180,E1 -7553.964,E2 -7553.964} C_VEL
LIN {X 0,Y 467.86,Z 230.208,A -85,B 0,C 180,E1 -7557.419,E2 -7557.419} C_VEL
LIN {X 0,Y 467.885,Z 230.206,A -85,B 0,C 180,E1 -7560.001,E2 -7560.001} C_VEL
LIN {X 0,Y 467.86,Z 230.207,A -85,B 0,C 180,E1 -7562.584,E2 -7562.584} C_VEL
LIN {X 0,Y 467.725,Z 230.225,A -85,B 0,C 180,E1 -7566.039,E2 -7566.039} C_VEL
LIN {X 0,Y 467.673,Z 230.23,A -85,B 0,C 180,E1 -7568.644,E2 -7568.644} C_VEL
LIN {X 0,Y 467.661,Z 230.231,A -85,B 0,C 180,E1 -7572.147,E2 -7572.147} C_VEL
LIN {X 0,Y 467.644,Z 230.235,A -85,B 0,C 180,E1 -7575.696,E2 -7575.696} C_VEL
LIN {X 0,Y 467.623,Z 230.236,A -85,B 0,C 180,E1 -7578.765,E2 -7578.765} C_VEL
LIN {X 0,Y 467.586,Z 230.243,A -85,B 0,C 180,E1 -7581.269,E2 -7581.269} C_VEL
LIN {X 0,Y 467.562,Z 230.244,A -85,B 0,C 180,E1 -7583.945,E2 -7583.945} C_VEL
LIN {X 0,Y 467.593,Z 230.241,A -85,B 0,C 180,E1 -7586.803,E2 -7586.803} C_VEL
LIN {X 0,Y 467.559,Z 230.246,A -85,B 0,C 180,E1 -7589.739,E2 -7589.739} C_VEL
LIN {X 0,Y 467.585,Z 230.242,A -85,B 0,C 180,E1 -7592.759,E2 -7592.759} C_VEL
LIN {X 0,Y 467.559,Z 230.244,A -85,B 0,C 180,E1 -7595.89,E2 -7595.89} C_VEL
LIN {X 0,Y 467.582,Z 230.244,A -85,B 0,C 180,E1 -7599.146,E2 -7599.146} C_VEL
LIN {X 0,Y 467.593,Z 230.239,A -85,B 0,C 180,E1 -7602.567,E2 -7602.567} C_VEL
LIN {X 0,Y 467.572,Z 230.242,A -85,B 0,C 180,E1 -7605.053,E2 -7605.053} C_VEL
LIN {X 0,Y 467.596,Z 230.241,A -85,B 0,C 180,E1 -7607.44,E2 -7607.44} C_VEL
LIN {X 0,Y 467.618,Z 230.381,A -85,B 0,C 180,E1 -7609.101,E2 -7609.101} C_VEL
LIN {X 0,Y 468.81,Z 236.972,A -85,B 0,C 180,E1 -7612.074,E2 -7612.074} C_VEL
LIN {X 0,Y 469.382,Z 241.363,A -85,B 0,C 180,E1 -7613.954,E2 -7613.954} C_VEL
LIN {X 0,Y 469.161,Z 247.309,A -85,B 0,C 180,E1 -7616.34,E2 -7616.34} C_VEL
LIN {X 0,Y 468.78,Z 255.196,A -85,B 0,C 180,E1 -7619.354,E2 -7619.354} C_VEL
LIN {X 0,Y 468.35,Z 264.408,A -85,B 0,C 180,E1 -7622.762,E2 -7622.762} C_VEL
LIN {X 0,Y 467.918,Z 273.711,A -85,B 0,C 180,E1 -7626.075,E2 -7626.075} C_VEL
LIN {X 0,Y 467.648,Z 283.335,A -85,B 0,C 180,E1 -7629.318,E2 -7629.318} C_VEL
LIN {X 0,Y 467.403,Z 291.538,A -85,B 0,C 180,E1 -7632.046,E2 -7632.046} C_VEL
LIN {X 0,Y 467.253,Z 299.195,A -85,B 0,C 180,E1 -7634.571,E2 -7634.571} C_VEL
LIN {X 0,Y 469.823,Z 314.733,A -85,B 0,C 180,E1 -7635.087,E2 -7635.087} C_VEL
LIN {X 0,Y 470.157,Z 319.572,A -85,B 0,C 180,E1 -7635.278,E2 -7635.278} C_VEL
LIN {X 0,Y 469.749,Z 331.245,A -85,B 0,C 180,E1 -7635.818,E2 -7635.818} C_VEL
LIN {X 0,Y 469.271,Z 342.473,A -85,B 0,C 180,E1 -7636.5,E2 -7636.5} C_VEL
LIN {X 0,Y 468.847,Z 352.99,A -85,B 0,C 180,E1 -7637.305,E2 -7637.305} C_VEL
LIN {X 0,Y 468.38,Z 363.592,A -85,B 0,C 180,E1 -7638.313,E2 -7638.313} C_VEL
LIN {X 0,Y 467.85,Z 372.782,A -85,B 0,C 180,E1 -7639.396,E2 -7639.396} C_VEL
LIN {X 0,Y 467.449,Z 381.685,A -85,B 0,C 180,E1 -7640.698,E2 -7640.698} C_VEL
LIN {X 0,Y 467.095,Z 388.846,A -85,B 0,C 180,E1 -7641.999,E2 -7641.999} C_VEL
LIN {X 0,Y 466.906,Z 395.092,A -85,B 0,C 180,E1 -7643.444,E2 -7643.444} C_VEL
LIN {X 0,Y 466.785,Z 399.675,A -85,B 0,C 180,E1 -7644.817,E2 -7644.817} C_VEL
LIN {X 0,Y 466.664,Z 401.956,A -85,B 0,C 180,E1 -7645.681,E2 -7645.681} C_VEL
LIN {X 0,Y 466.696,Z 403.806,A -85,B 0,C 180,E1 -7646.546,E2 -7646.546} C_VEL
LIN {X 0,Y 466.648,Z 405.192,A -85,B 0,C 180,E1 -7647.41,E2 -7647.41} C_VEL
LIN {X 0,Y 466.59,Z 406.785,A -85,B 0,C 180,E1 -7649.136,E2 -7649.136} C_VEL
LIN {X 0,Y 466.571,Z 407,A -85,B 0,C 180,E1 -7650,E2 -7650} C_VEL
LIN {X 0,Y 466.59,Z 406.786,A -85,B 0,C 180,E1 -7650.863,E2 -7650.863} C_VEL
LIN {X 0,Y 466.647,Z 405.196,A -85,B 0,C 180,E1 -7652.589,E2 -7652.589} C_VEL
LIN {X 0,Y 466.696,Z 403.811,A -85,B 0,C 180,E1 -7653.453,E2 -7653.453} C_VEL
LIN {X 0,Y 466.704,Z 400.896,A -85,B 0,C 180,E1 -7654.75,E2 -7654.75} C_VEL
LIN {X 0,Y 466.841,Z 396.95,A -85,B 0,C 180,E1 -7656.049,E2 -7656.049} C_VEL
LIN {X 0,Y 466.997,Z 390.878,A -85,B 0,C 180,E1 -7657.566,E2 -7657.566} C_VEL
LIN {X 0,Y 467.352,Z 384.238,A -85,B 0,C 180,E1 -7658.866,E2 -7658.866} C_VEL
LIN {X 0,Y 467.74,Z 375.995,A -85,B 0,C 180,E1 -7660.168,E2 -7660.168} C_VEL
LIN {X 0,Y 468.156,Z 367.523,A -85,B 0,C 180,E1 -7661.253,E2 -7661.253} C_VEL
LIN {X 0,Y 468.672,Z 357.195,A -85,B 0,C 180,E1 -7662.319,E2 -7662.319} C_VEL
LIN {X 0,Y 469.086,Z 345.555,A -85,B 0,C 180,E1 -7663.284,E2 -7663.284} C_VEL
LIN {X 0,Y 469.643,Z 333.216,A -85,B 0,C 180,E1 -7664.073,E2 -7664.073} C_VEL
LIN {X 0,Y 470.076,Z 320.84,A -85,B 0,C 180,E1 -7664.668,E2 -7664.668} C_VEL
LIN {X 0,Y 469.92,Z 315.466,A -85,B 0,C 180,E1 -7664.881,E2 -7664.881} C_VEL
LIN {X 0,Y 467.7,Z 302.421,A -85,B 0,C 180,E1 -7665.329,E2 -7665.329} C_VEL
LIN {X 0,Y 467.213,Z 299.102,A -85,B 0,C 180,E1 -7665.43,E2 -7665.43} C_VEL
LIN {X 0,Y 467.485,Z 289.063,A -85,B 0,C 180,E1 -7668.714,E2 -7668.714} C_VEL
